// Device/Application/Bausteine/SMB2_Client/NTLM/Functions/ProcessChallengeMessage
FUNCTION_BLOCK ProcessChallengeMessage
VAR_INPUT
	xExecute:BOOL; // Start
	session:POINTER TO SessionData; // NTLM Parameter
	challMess:POINTER TO CHALLENGE_MESSAGE; // Challenge Message
END_VAR
VAR_OUTPUT
	xDone:BOOL;
END_VAR
VAR
	timestamp:ARRAY[0..7] OF BYTE:= [ 16#C2,16#E8,16#2C,16#F5,16#9C,16#6D,16#D3,16#01];
	step:INT;
	clientChall:ARRAY[0..7] OF BYTE:= [16#bf, 16#c5, 16#f2, 16#3e, 16#c8, 16#82, 16#ba, 16#f1];//[16#9E, 16#B9, 16#86, 16#EC, 16#C3, 16#FE, 16#0F, 16#72]; //[16#87, 16#05, 16#42, 16#8E, 16#2A, 16#A3, 16#5D, 16#26];
	servertest:ARRAY[0..7] OF BYTE:= [16#0E, 16#CB, 16#9E, 16#63, 16#6E, 16#3E, 16#08, 16#50];
	NTOWFv2:NTOWFv2;
	LMOWFv2:LMOWFv2;
	SIGNKEY:SIGNKEY;
	SEALKEY:SEALKEY;
	mechListMic:mechListMic;
	ComputeResponse:ComputeResponse;
END_VAR

// Compute the whole Challenge Message and copy all results to session

xDone:=FALSE;
if step=0 and xExecute then
	step:=1;
END_IF

CASE step OF
1:	session^.serverChallenge := challMess^.ServerChallenge;
	session^.clientChallenge := clientChall;
	session^.NegotiateFlags := 16#E2880215;//challMess^.NegotiateFlags;
	step:=2;
	
	// Response Keys
2:	NTOWFv2(Passwd:=session^.password,User:=session^.user,UserDom:=session^.userDomain,out=>session^.responseKeyNT);
	NTOWFv2.xExecute:= TRUE;
	IF NTOWFv2.xDone THEN step:=step+1; END_IF
3:	LMOWFv2(Passwd:=session^.password,User:=session^.user,UserDom:=session^.userDomain,out=>session^.responseKeyLM);
	LMOWFv2.xExecute:= TRUE;
	IF LMOWFv2.xDone THEN step:=step+1; END_IF

	// Timestamp from Challenge Message
4: 	timestamp:= challMess^.AVPairList.TimeStamp;
	//challMess^.AVPairList.TimeStamp:=timestamp;
	step:=step+1;
	
5:	ComputeResponse(session:=session,challMess:=challMess,Timee:=timeStamp); // Compute NTProofStr, lmResponse, ntResponse, session base key
	ComputeResponse.xExecute:=TRUE;
	IF ComputeResponse.xDone THEN step:=step+1; END_IF

	// KeyExchange Key
6:	session^.keyExchangeKey:= session^.sessionBaseKey;
	step:=step+1;

7: 	// Encrypted Session Key
	EncryptedSessionKey(session:=session);
	step:=step+1;
	
	// Sign & Seal Keys
8:	SIGNKEY(ExportedSessionKey:=session^.exportedSessionKey,NegFlg:=session^.NegotiateFlags,Mode:=1,SignKey=>session^.ClientSigningKey);
	SIGNKEY.xExecute:=TRUE;
	IF SIGNKEY.xDone THEN SIGNKEY.xExecute:=FALSE; step:=step+1; END_IF
	
9:	SIGNKEY(ExportedSessionKey:=session^.exportedSessionKey,NegFlg:=session^.NegotiateFlags,Mode:=2,SignKey=>session^.ServerSigningKey);
	SIGNKEY.xExecute:=TRUE;
	IF SIGNKEY.xDone THEN SIGNKEY.xExecute:=FALSE; step:=step+1; END_IF
	
10:	SEALKEY(ExportedSessionKey:=session^.exportedSessionKey,NegFlg:=session^.NegotiateFlags,Mode:=1,SealKey=>session^.ClientSealingKey);
	SEALKEY.xExecute:=TRUE;
	IF SEALKEY.xDone THEN SEALKEY.xExecute:=FALSE; step:=step+1; END_IF
	
11:	SEALKEY(ExportedSessionKey:=session^.exportedSessionKey,NegFlg:=session^.NegotiateFlags,Mode:=2,SealKey=>session^.ServerSealingKey);
	SEALKEY.xExecute:=TRUE;
	IF SEALKEY.xDone THEN SEALKEY.xExecute:=FALSE; step:=step+1; END_IF

12:	mechListMic(session:=session,out=>session^.mechListMIC);
	mechListMic.xExecute:=TRUE;
	IF mechListMic.xDone THEN SEALKEY.xExecute:=FALSE; step:=step+1; END_IF
	
	// RC4 Init
13:	session^.clientHandle(key:=ADR(session^.ClientSealingKey),lenKey:=16,Mode:=0);
	session^.ServerHandle(key:=ADR(session^.ServerSealingKey),lenKey:=16,Mode:=0);
	xDone:=TRUE;
	step:=0;
	
END_CASE

END_FUNCTION_BLOCK

// Device/Application/Bausteine/SMB2_Client/NTLM/Functions/NTOWFv2
FUNCTION_BLOCK NTOWFv2
VAR_INPUT
	xExecute:BOOL;
	Passwd:WSTRING;
	User:WSTRING;
	UserDom:WSTRING;
END_VAR
VAR_OUTPUT
	xDone:BOOL;
	out:ARRAY[0..15] OF BYTE;
END_VAR
VAR
	Step:INT:=0;
	temp:ARRAY[0..15] OF BYTE:= [16#DD, 16#D0,16#B7,16#46,16#5E,16#B8,16#39,16#32,16#66,16#98,16#3F,16#B8,16#4D,16#7B,16#AD,16#9D];;
	concat:WSTRING;
	MD4:MD4;
	HMACMD5:HMAC_MD5;
END_VAR

(*
[MS-NLMP]
NTOWFv2(Passwd, User, UserDom) as HMAC_MD5( MD4(UNICODE(Passwd)), UNICODE(ConcatenationOf( Uppercase(User), UserDom ) ) )
*)

xDone := FALSE;
IF Step = 0 AND xExecute = 1 THEN
	Step:=1;
END_IF

CASE Step OF
0: 	xDone := FALSE;

1:	MD4(PT:=ADR(Passwd),Length:=(WLEN(Passwd)*2),digest=>temp); //MD4(UNICODE(Passwd))
	concat:= WCONCAT(WSTRING_UPPER(User),UserDom); // UNICODE(ConcatenationOf( Uppercase(User), UserDom )
	Step := 2;
	
2:	HMACMD5(key:=ADR(temp),lenKey:=16,message:=ADR(concat),lenMess:=WLEN(concat)*2,out=>out); // Hash HMAC_MD5( MD4(UNICODE(Passwd)), UNICODE(ConcatenationOf( Uppercase(User), UserDom ) ) )
	HMACMD5.xExecute:= TRUE;
	
	IF HMACMD5.xDone THEN
		HMACMD5.xExecute:= TRUE;	
		xDone := TRUE;
		Step:=0;
	END_IF
END_CASE

END_FUNCTION_BLOCK

// Device/Application/Bausteine/SMB2_Client/NTLM/Functions/Hash/Encryption/MD4
FUNCTION_BLOCK MD4
VAR_INPUT
	PT: POINTER TO ARRAY[0..127]OF BYTE;
	Length:INT;
END_VAR
VAR_OUTPUT
	digest:ARRAY[0..15] OF byte;
END_VAR
VAR
	A:UDINT:= 16#67452301;
	AA:UDINT:=0;
	B:UDINT:= 16#EFCDAB89; 
	BB:UDINT:=0;
	C:UDINT:= 16#98BADCFE; 
	CC:UDINT:=0;
	D:UDINT:= 16#10325476;
	DD:UDINT:=0;
	i:INT;
	j:INT;
	M:ARRAY[0..127] OF BYTE;
	MM:ARRAY[0..31] OF UDINT;
	X:ARRAY[0..15] OF UDINT;
	Len:INT;
	pVar:POINTER TO ARRAY[0..127] OF BYTE;
	pVar2:POINTER TO BYTE;
END_VAR

	A:=16#67452301;
	B:= 16#EFCDAB89; 
	C:= 16#98BADCFE; 
	D:= 16#10325476;
	
FOR i:=0 TO Length-1 DO
	M[i]:= PT^[i];
END_FOR
	// Apped 1 Bit to the Message
	M[Length] := 16#80;
	
	pVar:=ADR(M[0]);
	pVar2:=ADR(MM[0]);
	FOR i:=0 TO ((len+1)*64)-1 DO
		pVar2^:=pVar^[i];
		pVar2:=pVar2+1;
	END_FOR
	
	
IF Length < 64 THEN
	MM[14]:= INT_TO_UDINT(Length*8);
	len:=0;
ELSIF Length >= 64 AND Length < 128 THEN
	MM[30]:= INT_TO_UDINT(Length*8);
	len:=1;
END_IF	

	
FOR i:=0 TO len DO
	// Copy block i into X
	FOR j:=0 TO 15 DO
		X[j]:= MM[16*i+j];
	END_FOR
	 
	AA:=A;
	BB:=B;
	CC:=C;
	DD:=D;
	
	A:= ROUND1(A,B,C,D,X[0],3);
	D:=	ROUND1(D,A,B,C,X[1],7);
	C:=	ROUND1(C,D,A,B,X[2],11);
	B:=	ROUND1(B,C,D,A,X[3],19);
	A:=	ROUND1(A,B,C,D,X[4],3);
	D:=	ROUND1(D,A,B,C,X[5],7);
	C:=	ROUND1(C,D,A,B,X[6],11);
	B:=	ROUND1(B,C,D,A,X[7],19);
	A:=	ROUND1(A,B,C,D,X[8],3);
	D:=	ROUND1(D,A,B,C,X[9],7);
	C:=	ROUND1(C,D,A,B,X[10],11);
	B:=	ROUND1(B,C,D,A,X[11],19);
	A:=	ROUND1(A,B,C,D,X[12],3);
	D:=	ROUND1(D,A,B,C,X[13],7);
	C:=	ROUND1(C,D,A,B,X[14],11);
	B:=	ROUND1(B,C,D,A,X[15],19);
	
	A:=	ROUND2(A,B,C,D,X[0],3);
	D:=	ROUND2(D,A,B,C,X[4],5);
	C:=	ROUND2(C,D,A,B,X[8],9);
	B:=	ROUND2(B,C,D,A,X[12],13);
	A:=	ROUND2(A,B,C,D,X[1],3);
	D:=	ROUND2(D,A,B,C,X[5],5);
	C:=	ROUND2(C,D,A,B,X[9],9);
	B:=	ROUND2(B,C,D,A,X[13],13);
	A:=	ROUND2(A,B,C,D,X[2],3);
	D:=	ROUND2(D,A,B,C,X[6],5);
	C:=	ROUND2(C,D,A,B,X[10],9);
	B:=	ROUND2(B,C,D,A,X[14],13);
	A:=	ROUND2(A,B,C,D,X[3],3);
	D:=	ROUND2(D,A,B,C,X[7],5);
	C:=	ROUND2(C,D,A,B,X[11],9);
	B:=	ROUND2(B,C,D,A,X[15],13);
 
	A:=	ROUND3(A,B,C,D,X[0],3);
	D:=	ROUND3(D,A,B,C,X[8],9);
	C:=	ROUND3(C,D,A,B,X[4],11);
	B:=	ROUND3(B,C,D,A,X[12],15);
	A:=	ROUND3(A,B,C,D,X[2],3);
	D:=	ROUND3(D,A,B,C,X[10],9);
	C:=	ROUND3(C,D,A,B,X[6],11);
	B:=	ROUND3(B,C,D,A,X[14],15);
	A:=	ROUND3(A,B,C,D,X[1],3);
	D:=	ROUND3(D,A,B,C,X[9],9);
	C:=	ROUND3(C,D,A,B,X[5],11);
	B:=	ROUND3(B,C,D,A,X[13],15);
	A:=	ROUND3(A,B,C,D,X[3],3);
	D:=	ROUND3(D,A,B,C,X[11],9);
	C:=	ROUND3(C,D,A,B,X[7],11);
	B:=	ROUND3(B,C,D,A,X[15],15);
	
	A:=A+AA;
	B:=B+BB;
	C:=C+CC;
	D:=D+DD;
END_FOR

	digest[0]:=UDINT_TO_BYTE(A); digest[1]:=UDINT_TO_BYTE(SHR(A,8)); digest[2]:=UDINT_TO_BYTE(SHR(A,16)); digest[3]:=UDINT_TO_BYTE(SHR(A,24)); 
	digest[4]:=UDINT_TO_BYTE(B); digest[5]:=UDINT_TO_BYTE(SHR(B,8)); digest[6]:=UDINT_TO_BYTE(SHR(B,16)); digest[7]:=UDINT_TO_BYTE(SHR(B,24)); 
	digest[8]:=UDINT_TO_BYTE(C); digest[9]:=UDINT_TO_BYTE(SHR(C,8)); digest[10]:=UDINT_TO_BYTE(SHR(C,16)); digest[11]:=UDINT_TO_BYTE(SHR(C,24)); 
	digest[12]:=UDINT_TO_BYTE(D); digest[13]:=UDINT_TO_BYTE(SHR(D,8)); digest[14]:=UDINT_TO_BYTE(SHR(D,16)); digest[15]:=UDINT_TO_BYTE(SHR(D,24)); 

FOR i:=0 TO 127 DO
	M[i] := 0;
END_FOR

METHOD ROUND1 : UDINT
VAR_INPUT
	a:UDINT;
	b:UDINT;
	c:UDINT;
	d:UDINT;
	x:UDINT;
	ss:UDINT;
END_VAR
VAR
	temp:UDINT;
	temp1:UDINT;
	temp2:udint;
END_VAR
//#define F(X,Y,Z) (((X)&(Y))|((~(X))&(Z)))
//#define G(X,Y,Z) (((X)&(Y))|((X)&(Z))|((Y)&(Z)))
//#define H(X,Y,Z) ((X)^(Y)^(Z))
 
//#define LEFTROTATE(A,N) ((A)<<(N))|((A)>>(32-(N)))
 
//#define MD4ROUND1(a,b,c,d,x,s) a += F(b,c,d) + x; a = LEFTROTATE(a, s);
//#define MD4ROUND2(a,b,c,d,x,s) a += G(b,c,d) + x + (uint32_t)0x5A827999; a = LEFTROTATE(a, s);
//#define MD4ROUND3(a,b,c,d,x,s) a += H(b,c,d) + x + (uint32_t)0x6ED9EBA1; a = LEFTROTATE(a, s);

temp:= a  ;
temp1:=(((b AND c) OR ((NOT b) AND d))) ;
temp2:= x;

temp1:= temp+temp1;
temp:= temp1 + temp2;
ROUND1:= ROL(temp, ss);
END_METHOD

METHOD ROUND2 : UDINT
VAR_INPUT
	a:UDINT;
	b:UDINT;
	c:UDINT;
	d:UDINT;
	x:UDINT;
	ss:UDINT;
END_VAR
VAR
	temp:UDINT;
END_VAR
//#define F(X,Y,Z) (((X)&(Y))|((~(X))&(Z)))
//#define G(X,Y,Z) (((X)&(Y))|((X)&(Z))|((Y)&(Z)))
//#define H(X,Y,Z) ((X)^(Y)^(Z))
 
//#define LEFTROTATE(A,N) ((A)<<(N))|((A)>>(32-(N)))
 
//#define MD4ROUND1(a,b,c,d,x,s) a += F(b,c,d) + x; a = LEFTROTATE(a, s);
//#define MD4ROUND2(a,b,c,d,x,s) a += G(b,c,d) + x + (uint32_t)0x5A827999; a = LEFTROTATE(a, s);
//#define MD4ROUND3(a,b,c,d,x,s) a += H(b,c,d) + x + (uint32_t)0x6ED9EBA1; a = LEFTROTATE(a, s);

temp:= a + (((b)AND(c))OR((b)AND(d))OR((c)AND(d))) + x + 16#5A827999;

ROUND2:= ROL(temp, ss);
END_METHOD

METHOD ROUND3 : UDINT
VAR_INPUT
	a:UDINT;
	b:UDINT;
	c:UDINT;
	d:UDINT;
	x:UDINT;
	ss:UDINT;
END_VAR
VAR
	temp:UDINT;
END_VAR
//#define F(X,Y,Z) (((X)&(Y))|((~(X))&(Z)))
//#define G(X,Y,Z) (((X)&(Y))|((X)&(Z))|((Y)&(Z)))
//#define H(X,Y,Z) ((X)^(Y)^(Z))
 
//#define LEFTROTATE(A,N) ((A)<<(N))|((A)>>(32-(N)))
 
//#define MD4ROUND1(a,b,c,d,x,s) a += F(b,c,d) + x; a = LEFTROTATE(a, s);
//#define MD4ROUND2(a,b,c,d,x,s) a += G(b,c,d) + x + (uint32_t)0x5A827999; a = LEFTROTATE(a, s);
//#define MD4ROUND3(a,b,c,d,x,s) a += H(b,c,d) + x + (uint32_t)0x6ED9EBA1; a = LEFTROTATE(a, s);

temp:= a + ((b)XOR(c)XOR(d)) + x + 16#6ED9EBA1;

ROUND3:= ROL(temp, ss);
END_METHOD

END_FUNCTION_BLOCK

// Device/Application/Bausteine/SMB2_Client/Misc/WSTRING_UPPER
FUNCTION WSTRING_UPPER : WSTRING(80)
VAR_INPUT
	In:WSTRING(80);
END_VAR
VAR
	i:int;
	len:INT;
	pIn:POINTER TO ARRAY[0..79] OF WORD;
	pOut:POINTER TO ARRAY[0..79] OF WORD;
END_VAR

len:=wlen(In);

pIn:= ADR(In);
pOut:= ADR(WSTRING_UPPER);

FOR i:=0 TO len DO
	IF pIn^[i] >= 16#0061 AND pIn^[i] <= 16#007A THEN
		pOut^[i] := pIn^[i] - 16#0020;
	ELSE
		pOut^[i]:=pIn^[i]; 
	END_IF
END_FOR

END_FUNCTION

// Device/Application/Bausteine/SMB2_Client/NTLM/Functions/LMOWFv2
FUNCTION_BLOCK LMOWFv2
VAR_INPUT
	xExecute:BOOL;
	Passwd:WSTRING;
	User:WSTRING;
	UserDom:WSTRING;
END_VAR
VAR_OUTPUT
	xDone:BOOL;
	out:ARRAY[0..15] OF BYTE;
END_VAR
VAR
	NTOWFv2:NTOWFv2;
END_VAR

(*
[MS-NLMP]
LMOWFv2(Passwd, User, UserDom) as NTOWFv2(Passwd, User, UserDom)
*)

NTOWFv2(xExecute:= xExecute,Passwd:=Passwd,User:=User,UserDom:=UserDom,xDone=>xDone,out=>out);

END_FUNCTION_BLOCK

// Device/Application/Bausteine/SMB2_Client/NTLM/Functions/ComputeResponse
FUNCTION_BLOCK ComputeResponse
VAR_INPUT
	xExecute:BOOL; // Start
	session:POINTER TO sessionData; // NTLM Parameter
	challMess:POINTER TO CHALLENGE_MESSAGE; // Challenge Message
	Timee:ARRAY[0..7] OF BYTE; // Timestamp from Challenge Message
END_VAR
VAR_OUTPUT
	xDone:BOOL;
END_VAR
VAR
	Step:INT:=0;
	i:INT;
	temp:ARRAY[0..511] OF BYTE;
	tempLen:INT;
	pVar:POINTER TO ARRAY[0..32767] OF BYTE;
	ntProofStr:ARRAY[0..15] OF BYTE;
	temp2:ARRAY[0..511] OF BYTE;
	tempLen2:INT;
	hmacTemp:ARRAY[0..15] OF BYTE;
	HMACMD5:HMAC_MD5;

END_VAR

(*
	[MS-NLMP]
	Set temp to ConcatenationOf(Responserversion, HiResponserversion, Z(6), Time, ClientChallenge, Z(4), ServerName, Z(4)) 
	Set NTProofStr to HMAC_MD5(ResponseKeyNT, ConcatenationOf(CHALLENGE_MESSAGE.ServerChallenge,temp)) 
	Set NtChallengeResponse to ConcatenationOf(NTProofStr, temp) 
	Set LmChallengeResponse to ConcatenationOf(HMAC_MD5(ResponseKeyLM, ConcatenationOf(CHALLENGE_MESSAGE.ServerChallenge, ClientChallenge)), ClientChallenge )
*)

xDone:=FALSE;
IF Step = 0 AND xExecute = TRUE THEN
	Step:=1;
END_IF

CASE step OF
0:	
1:	//ConcatenationOf(Responserversion, HiResponserversion, Z(6), Time, ClientChallenge, Z(4), AVPairList, Z(4)) // Servername in NLMP Kap 3.3.1 means AVPairList
	i:=0;
	pVar:=ADR(temp);
	
	tempLen2 :=SetAVPairList(AVPairList:=challMess^.AVPairList,pOut:=ADR(temp2));
	
	FOR i:=0 TO 1 DO
		pVar^[i]:= 16#01;
	END_FOR
	FOR i:=i TO 1+6 DO
		pVar^[i]:= 16#00;
	END_FOR
	FOR i:=i TO 1+6+8 DO
		pVar^[i] := timee[i-(1+1+6)];
	END_FOR
	FOR i:=i TO 1+6+8+8 DO
		pVar^[i] :=	session^.clientChallenge[i-(1+1+6+8)];
	END_FOR
	FOR i:=i TO 1+6+8+8+4 DO
		pVar^[i]:= 16#00;
	END_FOR
	FOR i:=i TO 1+6+8+8+4+tempLen2 DO
		pVar^[i]:= temp2[i-(1+1+6+8+8+4)];
	END_FOR
	FOR i:=i TO 1+6+8+8+4+tempLen2+4 DO
		pVar^[i]:= 16#00;
	END_FOR
	tempLen:=i;
	step:=step+1;
	
	// ConcatenationOf(serverchallenge, temp)
2:	FOR i:=0 TO 7 DO
		temp2[i] := session^.serverChallenge[i];
	END_FOR
	FOR i:=i TO 7+tempLen DO
		temp2[i] := temp[i-(1+7)];
	END_FOR
	tempLen2:=i;
	step:=step+1;
	
	// NTProofStr = HMAC_MD5(responseKeyNt, temp2)
3:	HMACMD5(key:=ADR(session^.responseKeyNT),lenKey:=16 ,message:=ADR(temp2[0]), lenMess:=tempLen2+4,out=>ntProofStr); //<-- +4
	HMACMD5.xExecute:= TRUE;
	
	IF HMACMD5.xDone THEN
		step:= 4;
		HMACMD5.xExecute:= FALSE;
	END_IF

	// ntChallengeResponse = concat(ntProofStr, temp)
4:	FOR i:=0 TO 15 DO
		session^.ntChallengeResponse[i] := ntProofStr[i];
	END_FOR
	FOR i:=i TO 15+tempLen DO
		session^.ntChallengeResponse[i] := temp[i-(1+15)];
	END_FOR
	session^.ntChallengeResponseLen := INT_TO_WORD(i)+4; //<-- +4
	step:=step+1;
	
	// n.lmChallengeResponse = concat(hmacMd5(n.responseKeyLM, concat(n.serverChallenge, n.clientChallenge)), n.clientChallenge)
5:	FOR i:=0 TO 7 DO
		temp2[i] := session^.serverChallenge[i];
	END_FOR
	FOR i:=i TO 7+8 DO
		temp2[i] := session^.clientChallenge[i-8];
	END_FOR
	step:=step+1;
	
6: 	HMACMD5(key:=ADR(session^.responseKeyLM),lenKey:=16 ,message:=ADR(temp2[0]), lenMess:=32,out=>hmacTemp);
	HMACMD5.xExecute:= TRUE;
	
	IF HMACMD5.xDone THEN
		step:= 7;
		HMACMD5.xExecute:= FALSE;
	END_IF
	
7:	// Concat lmChallengeResponse
	FOR i:=0 TO 15 DO
		session^.lmChallengeResponse[i] := hmacTemp[i];
	END_FOR
	FOR i:=i TO 15+8 DO
		session^.lmChallengeResponse[i] := session^.clientChallenge[i-15];
	END_FOR
	session^.lmChallengeResponseLen := INT_TO_WORD(i);
	step:=step+1;
	FOR i:=0 TO UINT_TO_INT(session^.lmChallengeResponseLen) -1 DO // Make lmChallengeResponse zero, not used
		session^.lmChallengeResponse[i]:= 0;
	END_FOR
	
	
	// sessionBaseKey = hmacMd5(responseKeyNT, ntProofStr)
8: 	HMACMD5(key:=ADR(session^.responseKeyNT),lenKey:=16 ,message:=ADR(ntProofStr[0]), lenMess:=16,out=>session^.sessionBaseKey);
	HMACMD5.xExecute:= TRUE;
	
	IF HMACMD5.xDone THEN
		step:= 0;
		HMACMD5.xExecute:= FALSE;
		xDone:=TRUE;
	END_IF
END_CASE

END_FUNCTION_BLOCK

// Device/Application/Bausteine/SMB2_Client/NTLM/Functions/SetAVPairList
FUNCTION SetAVPairList : int
VAR_INPUT
	AVPairList:AVPairList; // Extracted Attribute from Challenge Message
	pOut:POINTER TO ARRAY[0..32767] OF BYTE; // Pointer to Buffer or Payload Buffer
END_VAR
VAR
	step:INT:=1;
	pVar:POINTER TO ARRAY[0..511] OF BYTE;
	pVarLen:POINTER TO ARRAY[0..511] OF BYTE;
	i:INT:=0;
	j:INT:=0;
	tempLen:INT;
	identifier:BYTE;;
	flags:DWORD:=16#00000002;
	channelBindings:ARRAY[0..15] OF BYTE:=[0];
	restrictions:ARRAY[0..47] OF BYTE:=	[16#30, 16#00, 16#00, 16#00, 16#00, 16#00, 16#00, 16#00, 16#01, 16#00, 16#00, 16#00, 16#00, 16#20, 16#00, 16#00,
										16#1C, 16#3A, 16#00, 16#6B, 16#51, 16#EA, 16#FC, 16#D1, 16#83, 16#AE, 16#BE, 16#D7, 16#48, 16#1C, 16#34, 16#4D,
										16#1C, 16#13, 16#C4, 16#E4, 16#4C, 16#39, 16#E8, 16#B8, 16#05, 16#4C, 16#63, 16#41, 16#66, 16#FF, 16#57, 16#0D];
	target:WSTRING(80);
	cifs:WSTRING:="cifs/";
	endOfList:BOOL;
END_VAR

// Building a new AVPairList / Target Info for Auth Message

endOfList:=0;
WHILE endOfList = 0 DO
	CASE step OF
		
		1:	// NB Domain Name
			tempLen :=wlen(AVPairList.NBDomainName)*2;
			pVar := ADR(AVPairList.NBDomainName);
			identifier:= 16#02;
			step:=step+1;
		2:	// NB Computer Name
			tempLen :=wlen(AVPairList.NBComputerName)*2;
			pVar := ADR(AVPairList.NBComputerName);
			identifier:= 16#01;
			step:=step+1;
		3:	// DNS Domain Name
			tempLen :=wlen(AVPairList.DNSDomainName)*2;
			pVar := ADR(AVPairList.DNSDomainName);
			identifier:= 16#04;
			step:=step+1;
		4:	// DNS Computer Name
			tempLen :=wlen(AVPairList.DNSComputerName)*2;
			pVar := ADR(AVPairList.DNSComputerName);
			identifier:= 16#03;
			step:=step+1;
		5:	// Timestamp
			tempLen :=8;
			pVar := ADR(AVPairList.TimeStamp);
			identifier:= 16#07;
			step:=step+1;
		6:	// Flags
			tempLen :=4;
			pVar := ADR(flags);
			identifier:= 16#06;
			step:=step+1;
		7:	// Restrictions
			tempLen := 48;
			pVar := ADR(restrictions);
			identifier:= 16#08;
			step:=step+1;
		8:	// Channel Bindings
			tempLen :=16;
			pVar := ADR(channelBindings);
			identifier:= 16#0A;
			step:=step+1;
		9:	// Target Name
			target:=wconcat(cifs,AVPairList.NBComputerName);
			tempLen :=wlen(target)*2;
			pVar := ADR(target);
			identifier:= 16#09;
			step:=1;
			// End of List
			endOfList:=TRUE;
	END_CASE
	// Identifier 
	pOut^[i]:= identifier; pOut^[i+1]:= 16#00; 
	i:=i+2;
	// length
	pVarLen := ADR(tempLen);
	FOR j:=0 TO 1 DO
		pOut^[i] := pVarLen ^[j];
		i:=i+1;
	END_FOR
	// data
	FOR j:=0 TO tempLen-1 DO
		pOut^[i] := pVar^[j];
		i:=i+1;
	END_FOR
	
	IF endOfList THEN
		FOR j:=0 TO 3 DO
		pOut^[i] := 16#00;
		i:=i+1;
		END_FOR
		SetAVPairList:=i;
	END_IF
END_WHILE

END_FUNCTION

// Device/Application/Bausteine/SMB2_Client/NTLM/Functions/EncryptedSessionKey
FUNCTION EncryptedSessionKey : int
VAR_INPUT
	session:POINTER TO sessionData;
END_VAR
VAR
	i:INT;
	temp:ARRAY[0..15] OF BYTE:=[16#C7, 16#9A, 16#31, 16#B6, 16#8D, 16#B6, 16#4E, 16#3F, 16#84, 16#66, 16#BE, 16#A3, 16#B2, 16#22, 16#3B, 16#C1];
	RC4K:RC4;
	temp2:dword;
END_VAR

(*	[MS-NLMP]
	If (NTLMSSP_NEGOTIATE_KEY_EXCH flag is set in NegFlg AND (NTLMSSP_NEGOTIATE_SIGN OR NTLMSSP_NEGOTIATE_SEAL are set in NegFlg) ) 
		Set ExportedSessionKey to RC4K(KeyExchangeKey, AUTHENTICATE_MESSAGE.EncryptedRandomSessionKey) 
	Else 
		Set ExportedSessionKey to KeyExchangeKey 
	EndIf 
*)

	temp2:= session^.NegotiateFlags AND 16#40000000;
IF (session^.NegotiateFlags AND 16#40000000) = 16#40000000 THEN
	session^.exportedSessionKey:= temp;
	RC4K(key:=ADR(session^.keyExchangeKey),lenKey:=16,data:=ADR(session^.exportedSessionKey),lenData:=16,ciper:=ADR(session^.encryptedRandomSessionKey),Mode:=2);
ELSE
	session^.exportedSessionKey := session^.keyExchangeKey;
	FOR i:=0 TO 15 DO
		session^.encryptedRandomSessionKey[i] := 16#00;
	END_FOR
END_IF

END_FUNCTION

// Device/Application/Bausteine/SMB2_Client/NTLM/Functions/SIGNKEY
FUNCTION_BLOCK SIGNKEY
VAR_INPUT
	xExecute:BOOL; // Start
	ExportedSessionKey:ARRAY[0..15] OF BYTE; // Exported Session Key
	NegFlg:DWORD; // Negotiate Flags
	Mode:BYTE; // 1= Client Signing Key, 2= Server Signing Key
END_VAR
VAR_OUTPUT
	xDone:BOOL;
	SignKey:ARRAY[0..15] OF BYTE;
END_VAR
VAR
	Step:INT;
	pVar:POINTER TO ARRAY[0..255] OF BYTE;
	i:INT;
	temp:ARRAY[0..74] OF BYTE;
	hash: MEM.MD5;
END_VAR
VAR CONSTANT
	Client:STRING:='session key to client-to-server signing key magic constant';
	Server:STRING:='session key to server-to-client signing key magic constant';
END_VAR

// This Function generates the Signing key from ExportedSessionKey and static String

//MS-NLMP 3.4.5.2

IF Step = 0 AND xExecute = TRUE THEN
	Step:=1;
ELSE
	xDone:= FALSE;
END_IF

IF (NegFlg AND UDINT_TO_DWORD(16#00080000)) = 16#00080000 THEN // EXTENDED_SESSIONSECURITY flag
	IF Mode = 1 THEN
		CASE Step OF
		0:	xDone:= FALSE;
		1:	FOR i:=0 TO 15 DO
				temp[i]:= ExportedSessionKey[i];
			END_FOR
			pVar:= ADR(Client);
			FOR i:=16 TO 16+standard.LEN(Client) DO
				temp[i]:= pVar^[i-16];
			END_FOR
				temp[i]:=0;
			Step:=2;
		2:	hash(pMemoryBlock:=ADR(Temp[0]),udiNumberOfBytes:=INT_TO_UDINT(16+standard.LEN(Client)+1),abyDigest=>SignKey);
			hash.xExecute:= TRUE;
	
			IF hash.xDone THEN
				step:= 0;
				hash.xExecute:= FALSE;
				xDone:= TRUE;
			END_IF
		END_CASE
	END_IF
	IF Mode = 2 THEN
		CASE Step OF
		0:	xDone:= FALSE;
		1:	FOR i:=0 TO 15 DO
				temp[i]:= ExportedSessionKey[i];
			END_FOR
			pVar:= ADR(Server);
			FOR i:=16 TO 16+standard.LEN(Server) DO
				temp[i]:= pVar^[i-16];
			END_FOR
			temp[i]:=0;
			Step:=2;
		2:	hash(pMemoryBlock:=ADR(Temp[0]),udiNumberOfBytes:=INT_TO_UDINT(standard.LEN(Client)+16+1),abyDigest=>SignKey);
			hash.xExecute:= TRUE;
	
			IF hash.xDone THEN
				step:= 0;
				hash.xExecute:= FALSE;
				xDone:= TRUE;
			END_IF
		END_CASE
	END_IF
ELSE
	FOR i:=0 TO 15 DO
		SignKey[i]:=0;	
	END_FOR
	xDone:= TRUE;
END_IF

END_FUNCTION_BLOCK

// Device/Application/Bausteine/SMB2_Client/NTLM/Functions/SEALKEY
FUNCTION_BLOCK SEALKEY
VAR_INPUT
	xExecute:BOOL; // Start
	ExportedSessionKey:ARRAY[0..15] OF BYTE; // Exported Session Key
	NegFlg:DWORD; // Negotiate Flags
	Mode:BYTE; // 1= Client Sealing Key, 2= Server Sealing Key
END_VAR
VAR_OUTPUT
	xDone:BOOL;
	SealKey:ARRAY[0..15] OF BYTE;
END_VAR
VAR
	SealKeyLen:INT;
	Step:INT;
	pVar:POINTER TO ARRAY[0..255] OF BYTE;
	i:INT;
	temp:ARRAY[0..74] OF BYTE;
	hash: MEM.MD5;
END_VAR
VAR CONSTANT
	Client:STRING:='session key to client-to-server sealing key magic constant';
	Server:STRING:='session key to server-to-client sealing key magic constant';
END_VAR

// This Function generates the Sealkey from ExportedSessionKey and static String

//MS-NLMP 3.4.5.3

xDone:= FALSE;
IF Step = 0 AND xExecute = TRUE THEN
	Step:=1;
END_IF


IF (NegFlg AND UDINT_TO_DWORD(16#00080000)) = 16#00080000 THEN // EXTENDED_SESSIONSECURITY flag
	IF (NegFlg AND UDINT_TO_DWORD(16#20000000)) = 16#20000000 THEN // NTLMSSP_NEGOTIATE_128
		SealKeyLen:= 16;
	ELSIF (NegFlg AND UDINT_TO_DWORD(16#80000000)) = 16#80000000 THEN // NTLMSSP_NEGOTIATE_56
		SealKeyLen:= 7;
	ELSE 
		SealKeyLen:= 5;
	END_IF

	IF Mode = 1 THEN
		CASE Step OF
		0:	xDone:= FALSE;
		1:	FOR i:=0 TO SealKeyLen DO
				temp[i]:= ExportedSessionKey[i];
			END_FOR
			pVar:= ADR(Client);
			FOR i:=SealKeyLen TO SealKeyLen+standard.LEN(Client) DO
				temp[i]:= pVar^[i-16];
			END_FOR
			temp[i]:=0;
			Step:=2;
		2:	hash(pMemoryBlock:=ADR(Temp[0]),udiNumberOfBytes:=INT_TO_UDINT(SealKeyLen+standard.LEN(Client)+1),abyDigest=>SealKey);
			hash.xExecute:= TRUE;
	
			IF hash.xDone THEN
				step:= 0;
				hash.xExecute:= FALSE;
				xDone:= TRUE;
			END_IF
		END_CASE
	ELSE
		CASE Step OF
		0:	xDone:= FALSE;
		1:	FOR i:=0 TO SealKeyLen DO
				temp[i]:= ExportedSessionKey[i];
			END_FOR
			pVar:= ADR(Server);
			FOR i:=SealKeyLen TO SealKeyLen+standard.LEN(Server) DO
				temp[i]:= pVar^[i-16];
			END_FOR
			temp[i]:=0;
			Step:=2;
		2:	hash(pMemoryBlock:=ADR(Temp[0]),udiNumberOfBytes:=INT_TO_UDINT(SealKeyLen+standard.LEN(Server)+1),abyDigest=>SealKey);
			hash.xExecute:= TRUE;
	
			IF hash.xDone THEN
				step:= 0;
				hash.xExecute:= FALSE;
				xDone:= TRUE;
			END_IF
		END_CASE
	END_IF
ELSIF ((NegFlg AND UDINT_TO_DWORD(16#00000200)) = 16#00000200) OR	// LM KEY
		((NegFlg AND UDINT_TO_DWORD(16#00000040)) = 16#00000040) THEN // DATAGRAM

	IF (NegFlg AND UDINT_TO_DWORD(16#80000000)) = 16#80000000 THEN // NTLMSSP_NEGOTIATE_56
		FOR i:=0 TO 5 DO
			temp[i]:= ExportedSessionKey[i];
		END_FOR
		temp[7]:= 16#A0;
	ELSE
		FOR i:=0 TO 4 DO
			temp[i]:= ExportedSessionKey[i];
		END_FOR
		temp[5]:= 16#E5; temp[6]:= 16#38; temp[7]:= 16#B0;
	END_IF
	FOR i:=0 TO 15 DO
		SealKey[i]:=temp[i];	
	END_FOR
	Step:=0;
	xDone:= TRUE;
ELSE
	FOR i:=0 TO 15 DO
		SealKey[i]:=ExportedSessionKey[i];	
	END_FOR
	Step:=0;
	xDone:= TRUE;
END_IF

END_FUNCTION_BLOCK

// Device/Application/Bausteine/SMB2_Client/SMB2/Functions/Requests/TreeConnectReq
FUNCTION TreeConnectReq : int
VAR_INPUT
	Connection:POINTER TO Connection; // Connection Parameter
	pSend:POINTER TO ARRAY[0..32767] OF BYTE; // Pointer to Send Buffer
	pSize:POINTER TO CAA.SIZE; // Send Size
	SharePathName:WSTRING(256); // name of Sharepath
END_VAR
VAR
	TransportHeader:SMB2_Transport_Header;
	SMB2Header: SMB2_Header_Sync;
	SMB2TreeConnect:SMB2_TREE_CONNECT_Request;
	sendS:UINT;
	startIndex:UINT;
END_VAR

// This Function generates the Tree Connect Request

	// Increase Message ID
	Connection^.MessageID[0]:= Connection^.MessageID[0]+1;	
	// Create Header
	SMB2Header.ProtocolID[0]:= 16#FE; SMB2Header.ProtocolID[1]:= 16#53; SMB2Header.ProtocolID[2]:= 16#4D; SMB2Header.ProtocolID[3]:= 16#42; 
	SMB2Header.StructureSize := 64;
	SMB2Header.CreditCharge := 0;
	SMB2Header.Status := 0;
	SMB2Header.Command := Constants.TREE_CONNECT;
	SMB2Header.CreditRepReq := 1;
	SMB2Header.Flags:= 0;
	SMB2Header.Flags := 0;
	SMB2Header.NextCommand := 0;		
	SMB2Header.MessageID[0]:= Connection^.MessageID[0]; SMB2Header.MessageID[1]:= 0;
	SMB2Header.TreeID:= 0;
	SMB2Header.SessionID[0]:= Connection^.Session.SessionID[0]; SMB2Header.SessionID[1]:= Connection^.Session.SessionID[1];
	SMB2Header.Signature[0]:= 0; SMB2Header.Signature[1]:= 0; SMB2Header.Signature[2]:= 0; SMB2Header.Signature[3]:= 0;
	
	// Create Tree Connect Request
	SMB2TreeConnect.StructureSize:= 9;
	SMB2TreeConnect.Flags:=0;
	SMB2TreeConnect.PathOffset:= 64 + 8;
	SMB2TreeConnect.PathName := SharePathName;
	SMB2TreeConnect.PathLength := INT_TO_WORD(wlen(SMB2TreeConnect.PathName)*2);
	
	
	// Copy Data in SendBuffer
	sendS:=SIZEOF(SMB2_Transport_Header);
	(*Parse SMB2 Header*)
	startIndex:=sendS-1;
	sendS:=sendS+SIZEOF(SMB2Header);
	MEM.MemMove(pSource:=ADR(SMB2Header) , pDestination:=ADR(pSend^[startIndex]) ,uiNumberOfBytes:=SIZEOF(SMB2Header));
	
	(*Parse Tree Connect Request*)
	startIndex:=sendS-1;
	sendS:=sendS+WORD_TO_UINT(SMB2TreeConnect.StructureSize-1+SMB2TreeConnect.PathLength);
	MEM.MemMove(pSource:=ADR(SMB2TreeConnect) , pDestination:=ADR(pSend^[startIndex]) ,uiNumberOfBytes:=WORD_TO_UINT(SMB2TreeConnect.StructureSize)-1+SMB2TreeConnect.PathLength);
	
	(*Parse Transport Header*)
	TransportHeader.Zero := 16#00;
	TransportHeader.StreamProtocolLength := SHR(MEM.ReverseBYTEsInDWORD(sendS-SIZEOF(TransportHeader)),8);
		
	startIndex:=0;
	MEM.MemMove(pSource:=ADR(TransportHeader) , pDestination:=ADR(pSend^[startIndex]) ,uiNumberOfBytes:=SIZEOF(SMB2_Transport_Header)-1);
	
	(*Set Sendsize*)	
	pSize^:= sendS-1;

END_FUNCTION

// Device/Application/Bausteine/SMB2_Client/SMB2/Functions/Requests/CloseReq
FUNCTION CloseReq : int
VAR_INPUT
	Connection:POINTER TO Connection; // Connection Parameter
	pSend:POINTER TO ARRAY[0..32767] OF BYTE; // Pointer to Send Buffer
	pSize:POINTER TO CAA.SIZE; // Send Size
END_VAR
VAR
	i:INT;
	TransportHeader:SMB2_Transport_Header;
	SMB2Header: SMB2_Header_Sync;
	SMB2Close: SMB2_Close_Request;
	sendS:UINT;
	startIndex:UINT;
	pVar: POINTER TO ARRAY[0..255] OF BYTE;
END_VAR

// This Function generates the Close Request

	// Increase Message ID
	Connection^.MessageID[0]:= Connection^.MessageID[0]+1;	
	// Create Header
	SMB2Header.ProtocolID[0]:= 16#FE; SMB2Header.ProtocolID[1]:= 16#53; SMB2Header.ProtocolID[2]:= 16#4D; SMB2Header.ProtocolID[3]:= 16#42; 
	SMB2Header.StructureSize := 64;
	SMB2Header.CreditCharge := 0;
	SMB2Header.Status := 0;
	SMB2Header.Command := Constants.CLOSE;
	SMB2Header.CreditRepReq := 1;
	SMB2Header.Flags:= 0;
	SMB2Header.Flags := 0;
	SMB2Header.NextCommand := 0;		
	SMB2Header.MessageID[0]:= Connection^.MessageID[0]; SMB2Header.MessageID[1]:= 0;
	SMB2Header.TreeID:= connection^.Session.TreeConnect.TreeConnectId;
	SMB2Header.SessionID[0]:= Connection^.Session.SessionID[0]; SMB2Header.SessionID[1]:= Connection^.Session.SessionID[1];
	SMB2Header.Signature[0]:= 0; SMB2Header.Signature[1]:= 0; SMB2Header.Signature[2]:= 0; SMB2Header.Signature[3]:= 0;
	
	// Close Request
	SMB2Close.StructureSize := 24;
	SMB2Close.Flags:=0;
	SMB2Close.FileId := Connection[0].Session.Open.FileId;
	
	// Copy Data in SendBuffer
	sendS:=SIZEOF(SMB2_Transport_Header);
	(*Parse SMB2 Header*)
	startIndex:=sendS-1;
	sendS:=sendS+SIZEOF(SMB2Header);
	MEM.MemMove(pSource:=ADR(SMB2Header) , pDestination:=ADR(pSend^[startIndex]) ,uiNumberOfBytes:=SIZEOF(SMB2Header));
	
	(*Parse Close Request*)
	startIndex:=sendS-1;
	sendS:=sendS+WORD_TO_UINT(SMB2Close.StructureSize);
	MEM.MemMove(pSource:=ADR(SMB2Close) , pDestination:=ADR(pSend^[startIndex]) ,uiNumberOfBytes:=WORD_TO_UINT(SMB2Close.StructureSize));
	
	(*Parse Transport Header*)
	TransportHeader.Zero := 16#00;
	TransportHeader.StreamProtocolLength := SHR(MEM.ReverseBYTEsInDWORD(sendS-SIZEOF(TransportHeader)),8);
		
	startIndex:=0;
	MEM.MemMove(pSource:=ADR(TransportHeader) , pDestination:=ADR(pSend^[startIndex]) ,uiNumberOfBytes:=SIZEOF(SMB2_Transport_Header)-1);
	
	(*Set Sendsize*)	
	pSize^:= sendS-1;

END_FUNCTION

// Device/Application/Bausteine/SMB2_Client/SMB2/Functions/Requests/TreeDisconnectReq
FUNCTION TreeDisconnectReq : int
VAR_INPUT
	Connection:POINTER TO Connection; // Connection Parameter
	pSend:POINTER TO ARRAY[0..32767] OF BYTE; // Pointer to Send Buffer
	pSize:POINTER TO CAA.SIZE; // Send Size
END_VAR
VAR
	TransportHeader:SMB2_Transport_Header;
	SMB2Header: SMB2_Header_Sync;
	SMB2Dis: SMB2_TREE_DISCONNECT_Request;
	sendS:UINT;
	startIndex:UINT;
END_VAR

// This Function generates the Tree Disconnect Request

	// Increase Message ID
	Connection^.MessageID[0]:= Connection^.MessageID[0]+1;	
	// Create Header
	SMB2Header.ProtocolID[0]:= 16#FE; SMB2Header.ProtocolID[1]:= 16#53; SMB2Header.ProtocolID[2]:= 16#4D; SMB2Header.ProtocolID[3]:= 16#42; 
	SMB2Header.StructureSize := 64;
	SMB2Header.CreditCharge := 0;
	SMB2Header.Status := 0;
	SMB2Header.Command := Constants.TREE_DISCONNECT;
	SMB2Header.CreditRepReq := 1;
	SMB2Header.Flags:= 0;
	SMB2Header.Flags := 0;
	SMB2Header.NextCommand := 0;		
	SMB2Header.MessageID[0]:= Connection^.MessageID[0]; SMB2Header.MessageID[1]:= 0;
	SMB2Header.TreeID:= connection^.Session.TreeConnect.TreeConnectId;
	SMB2Header.SessionID[0]:= Connection^.Session.SessionID[0]; SMB2Header.SessionID[1]:= Connection^.Session.SessionID[1];
	SMB2Header.Signature[0]:= 0; SMB2Header.Signature[1]:= 0; SMB2Header.Signature[2]:= 0; SMB2Header.Signature[3]:= 0;
	
	// Tree Disconnect Request
	SMB2Dis.StructureSize := 4;
	SMB2Dis.Reserved := 0;
	
	// Copy Data in SendBuffer
	sendS:=SIZEOF(SMB2_Transport_Header);
	(*Parse SMB2 Header*)
	startIndex:=sendS-1;
	sendS:=sendS+SIZEOF(SMB2Header);
	MEM.MemMove(pSource:=ADR(SMB2Header) , pDestination:=ADR(pSend^[startIndex]) ,uiNumberOfBytes:=SIZEOF(SMB2Header));
	
	(*Parse Tree Disconnect Request*)
	startIndex:=sendS-1;
	sendS:=sendS+WORD_TO_UINT(SMB2Dis.StructureSize);
	MEM.MemMove(pSource:=ADR(SMB2Dis) , pDestination:=ADR(pSend^[startIndex]) ,uiNumberOfBytes:=WORD_TO_UINT(SMB2Dis.StructureSize));
	
	(*Parse Transport Header*)
	TransportHeader.Zero := 16#00;
	TransportHeader.StreamProtocolLength := SHR(MEM.ReverseBYTEsInDWORD(sendS-SIZEOF(TransportHeader)),8);
		
	startIndex:=0;
	MEM.MemMove(pSource:=ADR(TransportHeader) , pDestination:=ADR(pSend^[startIndex]) ,uiNumberOfBytes:=SIZEOF(SMB2_Transport_Header)-1);
	
	(*Set Sendsize*)	
	pSize^:= sendS-1;

END_FUNCTION

// Device/Application/Bausteine/SMB2_Client/SMB2/Functions/Requests/LogOffReq
FUNCTION LogOffReq : int
VAR_INPUT
	Connection:POINTER TO Connection; // Connection Parameter
	pSend:POINTER TO ARRAY[0..32767] OF BYTE; // Pointer to Send Buffer
	pSize:POINTER TO CAA.SIZE; // Send Size
END_VAR
VAR
	TransportHeader:SMB2_Transport_Header;
	SMB2Header: SMB2_Header_Sync;
	SMB2LogOff: SMB2_LOGOFF_Request;
	sendS:UINT;
	startIndex:UINT;
END_VAR

// This Function generates the LogOff Request

	// Increase Message ID
	Connection^.MessageID[0]:= Connection^.MessageID[0]+1;	
	// Create Header
	SMB2Header.ProtocolID[0]:= 16#FE; SMB2Header.ProtocolID[1]:= 16#53; SMB2Header.ProtocolID[2]:= 16#4D; SMB2Header.ProtocolID[3]:= 16#42; 
	SMB2Header.StructureSize := 64;
	SMB2Header.CreditCharge := 0;
	SMB2Header.Status := 0;
	SMB2Header.Command := Constants.LOGOFF;
	SMB2Header.CreditRepReq := 1;
	SMB2Header.Flags:= 0;
	SMB2Header.Flags := 0;
	SMB2Header.NextCommand := 0;		
	SMB2Header.MessageID[0]:= Connection^.MessageID[0]; SMB2Header.MessageID[1]:= 0;
	SMB2Header.TreeID:= 0;
	SMB2Header.SessionID[0]:= Connection^.Session.SessionID[0]; SMB2Header.SessionID[1]:= Connection^.Session.SessionID[1];
	SMB2Header.Signature[0]:= 0; SMB2Header.Signature[1]:= 0; SMB2Header.Signature[2]:= 0; SMB2Header.Signature[3]:= 0;
	
	// LogOff Request
	SMB2LogOff.StructureSize := 4;
	SMB2LogOff.Reserved := 0;
	
	// Copy Data in SendBuffer
	sendS:=SIZEOF(SMB2_Transport_Header);
	(*Parse SMB2 Header*)
	startIndex:=sendS-1;
	sendS:=sendS+SIZEOF(SMB2Header);
	MEM.MemMove(pSource:=ADR(SMB2Header) , pDestination:=ADR(pSend^[startIndex]) ,uiNumberOfBytes:=SIZEOF(SMB2Header));
	
	(*Parse LogOff Request*)
	startIndex:=sendS-1;
	sendS:=sendS+WORD_TO_UINT(SMB2LogOff.StructureSize);
	MEM.MemMove(pSource:=ADR(SMB2LogOff) , pDestination:=ADR(pSend^[startIndex]) ,uiNumberOfBytes:=WORD_TO_UINT(SMB2LogOff.StructureSize));
	
	(*Parse Transport Header*)
	TransportHeader.Zero := 16#00;
	TransportHeader.StreamProtocolLength := SHR(MEM.ReverseBYTEsInDWORD(sendS-SIZEOF(TransportHeader)),8);
		
	startIndex:=0;
	MEM.MemMove(pSource:=ADR(TransportHeader) , pDestination:=ADR(pSend^[startIndex]) ,uiNumberOfBytes:=SIZEOF(SMB2_Transport_Header)-1);
	
	(*Set Sendsize*)	
	pSize^:= sendS-1;

END_FUNCTION

// Device/Application/Bausteine/SMB2_Client/SMB2/Functions/Requests/CreateReq
FUNCTION CreateReq : int
VAR_INPUT
	Connection:POINTER TO Connection; // Connection Parameter
	pSend:POINTER TO ARRAY[0..32767] OF BYTE; // Pointer to Send Buffer
	pSize:POINTER TO CAA.SIZE; // Send Size
	fileName:WSTRING(256); // filename in SMB Server
	mode:INT; // 1= Send, 2= Receive, 3= Explorer (Dir/File Names), 4=srcsvc (Sharenames)
END_VAR
VAR
	i:INT;
	TransportHeader:SMB2_Transport_Header;
	SMB2Header: SMB2_Header_Sync;
	SMB2Create: SMB2_CREATE_Request;
	sendS:UINT;
	startIndex:UINT;
	pVar: POINTER TO ARRAY[0..255] OF BYTE;
	mode_3_length:WORD;
END_VAR

// This Function generates the Create Request

	// Increase Message ID
	Connection^.MessageID[0]:= Connection^.MessageID[0]+1;	
	// Create Header
	SMB2Header.ProtocolID[0]:= 16#FE; SMB2Header.ProtocolID[1]:= 16#53; SMB2Header.ProtocolID[2]:= 16#4D; SMB2Header.ProtocolID[3]:= 16#42; 
	SMB2Header.StructureSize := 64;
	SMB2Header.CreditCharge := 0;
	SMB2Header.Status := 0;
	SMB2Header.Command := Constants.CREATE;
	SMB2Header.CreditRepReq := 1;
	SMB2Header.Flags:= 0;
	SMB2Header.Flags := 0;
	SMB2Header.NextCommand := 0;		
	SMB2Header.MessageID[0]:= Connection^.MessageID[0]; SMB2Header.MessageID[1]:= 0;
	SMB2Header.TreeID:= connection^.Session.TreeConnect.TreeConnectId;
	SMB2Header.SessionID[0]:= Connection^.Session.SessionID[0]; SMB2Header.SessionID[1]:= Connection^.Session.SessionID[1];
	SMB2Header.Signature[0]:= 0; SMB2Header.Signature[1]:= 0; SMB2Header.Signature[2]:= 0; SMB2Header.Signature[3]:= 0;
	
	// Create Request
	SMB2Create.StructureSize:= 57;
	SMB2Create.SecurityFlags := 0;
	SMB2Create.RequestedOplockLevel := 16#08; // Named Pipe = 0
	SMB2Create.ImpersonationLevel := 2;
	SMB2Create.SmbCreateFlags[0] := 0; SMB2Create.SmbCreateFlags[1] := 0; // Must be 0
	SMB2Create.Reserved[0] := 0; SMB2Create.Reserved[1] := 0;
	IF mode = 1 THEN // Create new file or Open
		SMB2Create.DesiredAccess := 16#0017019F; // FILE_WRITE_DATA
		SMB2Create.FileAttributes := 16#00000020; // FILE_ATTRIBUTE_NORMAL
		SMB2Create.CreateDisposition := 16#00000005; // FILE_CREATE - If the file already exists, fail the operation; otherwise, create the file.
		SMB2Create.CreateOptions := 16#00000064;
		SMB2Create.ShareAccess := 0;	
	ELSIF mode = 2 THEN // Open File
		SMB2Create.DesiredAccess := 16#00100081; // 
		SMB2Create.FileAttributes := 16#00000000; // 
		SMB2Create.CreateDisposition := 16#00000001; // OPEN - if file exists open it, else fail
		SMB2Create.CreateOptions := 16#00000020;
		SMB2Create.ShareAccess := 16#00000007;	
	ELSIF mode = 3 THEN // Explorer
		SMB2Create.DesiredAccess := 16#00100081; // 
		SMB2Create.FileAttributes := 16#00000000; // 
		SMB2Create.CreateDisposition := 16#00000001; // OPEN - if file exists open it, else fail
		SMB2Create.CreateOptions := 16#00000020;
		SMB2Create.ShareAccess := 16#00000001;	
	ELSIF mode = 4 THEN // srvsvc
		SMB2Create.DesiredAccess := 16#0012019F; // 
		SMB2Create.FileAttributes := 16#00000000; // 
		SMB2Create.CreateDisposition := 16#00000001; // OPEN - if file exists open it, else fail
		SMB2Create.CreateOptions := 16#00000040;
		SMB2Create.ShareAccess := 16#00000007;	
	END_IF
	
	SMB2Create.NameOffset := 64+56;
	SMB2Create.NameLength := DINT_TO_WORD(wlen(fileName)*2);
	SMB2Create.CreateContextsLength := 0;
	SMB2Create.CreateContextsOffset := 0;
	pVar:=ADR(fileName);
	
	IF (WLEN(fileName) = 0) THEN // filename empty (explorer mode)
		SMB2Create.Payload[0]:= 0;
		SMB2Create.Payload[1]:= 0;
		mode_3_length:=2;
	ELSE
		FOR i:=0 TO WORD_TO_INT(SMB2Create.NameLength)-1 DO
		SMB2Create.Payload[i] := pVar^[i];
		mode_3_length:=0;
	END_FOR
		
	END_IF

	// Copy Data in SendBuffer
	sendS:=SIZEOF(SMB2_Transport_Header);
	(*Parse SMB2 Header*)
	startIndex:=sendS-1;
	sendS:=sendS+SIZEOF(SMB2Header);
	MEM.MemMove(pSource:=ADR(SMB2Header) , pDestination:=ADR(pSend^[startIndex]) ,uiNumberOfBytes:=SIZEOF(SMB2Header));
	
	(*Parse Create Request*)
	startIndex:=sendS-1;
	sendS:=sendS+WORD_TO_UINT(SMB2Create.StructureSize-1+SMB2Create.NameLength+mode_3_length);
	MEM.MemMove(pSource:=ADR(SMB2Create) , pDestination:=ADR(pSend^[startIndex]) ,uiNumberOfBytes:=WORD_TO_UINT(SMB2Create.StructureSize)-1+SMB2Create.NameLength+mode_3_length);
	
	(*Parse Transport Header*)
	TransportHeader.Zero := 16#00;
	TransportHeader.StreamProtocolLength := SHR(MEM.ReverseBYTEsInDWORD(sendS-SIZEOF(TransportHeader)),8);
		
	startIndex:=0;
	MEM.MemMove(pSource:=ADR(TransportHeader) , pDestination:=ADR(pSend^[startIndex]) ,uiNumberOfBytes:=SIZEOF(SMB2_Transport_Header)-1);
	
	(*Set Sendsize*)	
	pSize^:= sendS-1;

END_FUNCTION

// Device/Application/Bausteine/SMB2_Client/SMB2/Functions/Requests/QueryDirReq
FUNCTION QueryDirReq : int
VAR_INPUT
	Connection:POINTER TO Connection; // Connection Parameter
	pSend:POINTER TO ARRAY[0..32767] OF BYTE; // Pointer to Send Buffer
	pSize:POINTER TO CAA.SIZE; // Send Size
END_VAR
VAR
	i:INT;
	TransportHeader:SMB2_Transport_Header;
	SMB2Header: SMB2_Header_Sync;
	SMB2QueryDir: SMB2_QUERY_DIRECTORY_Request;
	sendS:UINT;
	startIndex:UINT;
	pVar: POINTER TO ARRAY[0..255] OF BYTE;
END_VAR

// This Function generates the Query Directory Request

	// Increase Message ID
	Connection^.MessageID[0]:= Connection^.MessageID[0]+1;	
	// Create Header
	SMB2Header.ProtocolID[0]:= 16#FE; SMB2Header.ProtocolID[1]:= 16#53; SMB2Header.ProtocolID[2]:= 16#4D; SMB2Header.ProtocolID[3]:= 16#42; 
	SMB2Header.StructureSize := 64;
	SMB2Header.CreditCharge := 0;
	SMB2Header.Status := 0;
	SMB2Header.Command := Constants.QUERY_DIRECTORY;
	SMB2Header.CreditRepReq := 1;
	SMB2Header.Flags:= 0;
	SMB2Header.Flags := 0;
	SMB2Header.NextCommand := 0;		
	SMB2Header.MessageID[0]:= Connection^.MessageID[0]; SMB2Header.MessageID[1]:= 0;
	SMB2Header.TreeID:= connection^.Session.TreeConnect.TreeConnectId;
	SMB2Header.SessionID[0]:= Connection^.Session.SessionID[0]; SMB2Header.SessionID[1]:= Connection^.Session.SessionID[1];
	SMB2Header.Signature[0]:= 0; SMB2Header.Signature[1]:= 0; SMB2Header.Signature[2]:= 0; SMB2Header.Signature[3]:= 0;
	
	// Query Directory Request
	SMB2QueryDir.StructureSize:= 33;
	SMB2QueryDir.FileInformationClass := 16#01; // Detailed information on the names of files and directories in a directory.
	SMB2QueryDir.Flags:= 0;
	SMB2QueryDir.FileIndex:=0;
	SMB2QueryDir.FileId:=Connection^.Session.Open.FileId;
	SMB2QueryDir.FileNameOffset:= 16#0060;
	SMB2QueryDir.FileNameLength:=2;
	SMB2QueryDir.OutputbufferLength:=8196;
	SMB2QueryDir.Payload[0]:= 16#2A; SMB2QueryDir.Payload[1]:= 16#00; // "*" für alles

	
	// Copy Data in SendBuffer
	sendS:=SIZEOF(SMB2_Transport_Header);
	(*Parse SMB2 Header*)
	startIndex:=sendS-1;
	sendS:=sendS+SIZEOF(SMB2Header);
	MEM.MemMove(pSource:=ADR(SMB2Header) , pDestination:=ADR(pSend^[startIndex]) ,uiNumberOfBytes:=SIZEOF(SMB2Header));
	
	(*Parse Query Directory Request*)
	startIndex:=sendS-1;
	sendS:=sendS+WORD_TO_UINT(SMB2QueryDir.StructureSize-1+SMB2QueryDir.FileNameLength);
	MEM.MemMove(pSource:=ADR(SMB2QueryDir) , pDestination:=ADR(pSend^[startIndex]) ,uiNumberOfBytes:=WORD_TO_UINT(SMB2QueryDir.StructureSize)-1+SMB2QueryDir.FileNameLength);
	
	(*Parse Transport Header*)
	TransportHeader.Zero := 16#00;
	TransportHeader.StreamProtocolLength := SHR(MEM.ReverseBYTEsInDWORD(sendS-SIZEOF(TransportHeader)),8);
		
	startIndex:=0;
	MEM.MemMove(pSource:=ADR(TransportHeader) , pDestination:=ADR(pSend^[startIndex]) ,uiNumberOfBytes:=SIZEOF(SMB2_Transport_Header)-1);
	
	(*Set Sendsize*)	
	pSize^:= sendS-1;

END_FUNCTION

// Device/Application/Bausteine/SMB2_Client/SMB2/Functions/NetShareBind
FUNCTION NetShareBind : int
VAR_INPUT
	Connection:POINTER TO Connection; // Connection Parameter
	pSend:POINTER TO ARRAY[0..32767] OF BYTE; // Pointer to Send Buffer
	pSize:POINTER TO CAA.SIZE; // Send Size
END_VAR
VAR
	i:INT;
	j:INT;
	TransportHeader:SMB2_Transport_Header;
	SMB2Header: SMB2_Header_Sync;
	SMB2Write: SMB2_WRITE_Request;
	sendS:UINT;
	startIndex:UINT;
	tempLWORD:LWORD;
	tempWORD:WORD;
	pVar: POINTER TO ARRAY[0..255] OF BYTE;
	tempwString:WSTRING;
	posFraglength:INT;
	posAllochint:INT;
	tempLenDRC:INT;
	srvsvcUID:ARRAY[0..15] OF BYTE:=[16#C8, 16#4F, 16#32, 16#4B, 16#70, 16#16, 16#D3, 16#01, 16#12, 16#78, 16#5A, 16#47, 16#BF, 16#6E, 16#E1, 16#88];
	ndrUID:ARRAY[0..15] OF BYTE:=[16#04, 16#5D, 16#88, 16#8A, 16#EB, 16#1C, 16#C9, 16#11, 16#9F, 16#E8, 16#08, 16#00, 16#2B, 16#10, 16#48, 16#60];
	ndrUIDV1:ARRAY[0..15] OF BYTE:=[16#33, 16#05, 16#71, 16#71, 16#BA, 16#BE, 16#37, 16#49, 16#83, 16#19, 16#B5, 16#DB, 16#EF, 16#9C, 16#CC, 16#36];
	bindUID:ARRAY[0..15] OF BYTE:=[16#2C, 16#1C, 16#B7, 16#6C, 16#12, 16#98, 16#40, 16#45, 16#03, 16#00, 16#00, 16#00, 16#00, 16#00, 16#00, 16#00];
END_VAR

// This function generates the NetShareBind, function is unknown, all Values and the Structure is copied from Wireshark

	// Increase Message ID
	Connection^.MessageID[0]:= Connection^.MessageID[0]+1;	
	// Create Header
	SMB2Header.ProtocolID[0]:= 16#FE; SMB2Header.ProtocolID[1]:= 16#53; SMB2Header.ProtocolID[2]:= 16#4D; SMB2Header.ProtocolID[3]:= 16#42; 
	SMB2Header.StructureSize := 64;
	SMB2Header.CreditCharge := 0;
	SMB2Header.Status := 0;
	SMB2Header.Command := Constants.write;
	SMB2Header.CreditRepReq := 1;
	SMB2Header.Flags:= 0;
	SMB2Header.Flags := 0;
	SMB2Header.NextCommand := 0;		
	SMB2Header.MessageID[0]:= Connection^.MessageID[0]; SMB2Header.MessageID[1]:= 0;
	SMB2Header.TreeID:= connection^.Session.TreeConnect.TreeConnectId;
	SMB2Header.SessionID[0]:= Connection^.Session.SessionID[0]; SMB2Header.SessionID[1]:= Connection^.Session.SessionID[1];
	SMB2Header.Signature[0]:= 0; SMB2Header.Signature[1]:= 0; SMB2Header.Signature[2]:= 0; SMB2Header.Signature[3]:= 0;
	
	// Write, all these values are copied from Wireshark
	SMB2Write.StructureSize:=16#0031;
	SMB2Write.DataOffset:=16#0070;
	SMB2Write.Length:=160;
	SMB2Write.Offset:=0;
	SMB2Write.FileId:= Connection[0].Session.Open.FileId;
	SMB2Write.Channel:=0;
	SMB2Write.WriteChannelInfoLength:=0;
	SMB2Write.RemainingBytes:=0;
	SMB2Write.Flags:=0;
	
	//Build DCE/RPC
	
	i:=16#70+4;
	
	pSend^[i]:=16#05; i:=i+1; // Version 5
	pSend^[i]:=16#00; i:=i+1; // Version Minor 0 -> 5.0
	pSend^[i]:=16#0B; i:=i+1; // Request Type (Bind)
	pSend^[i]:=16#03; i:=i+1; // Flags
	pSend^[i]:=16#10; i:=i+1; pSend^[i]:=16#00; i:=i+1; pSend^[i]:=16#00; i:=i+1; pSend^[i]:=16#00; i:=i+1; // Data Represantation (Little Endian, Char: ASCII, Float: IEEE)
	pSend^[i]:=16#A0; i:=i+1; pSend^[i]:=16#00; i:=i+1; // Frag Length
	pSend^[i]:=16#00; i:=i+1; pSend^[i]:=16#00; i:=i+1; // Auth Length
	pSend^[i]:=16#02; i:=i+1; pSend^[i]:=16#00; i:=i+1; pSend^[i]:=16#00; i:=i+1; pSend^[i]:=16#00; i:=i+1; // Call ID
	pSend^[i]:=16#B8; i:=i+1; pSend^[i]:=16#10; i:=i+1; // Max Xmit Frag
	pSend^[i]:=16#B8; i:=i+1; pSend^[i]:=16#10; i:=i+1; // Max Receive Frag
	pSend^[i]:=16#00; i:=i+1; pSend^[i]:=16#00; i:=i+1; pSend^[i]:=16#00; i:=i+1; pSend^[i]:=16#00; i:=i+1; // Asoc Group
	pSend^[i]:=16#03; i:=i+1; // Num Ctx Items - 3
	pSend^[i]:=16#00; i:=i+1; pSend^[i]:=16#00; i:=i+1; pSend^[i]:=16#00; i:=i+1; // Padding 3 bytes
	
	// Ctx Item 1
	pSend^[i]:=16#00; i:=i+1; pSend^[i]:=16#00; i:=i+1; // Context ID
	pSend^[i]:=16#01; i:=i+1; // Num Trans Items
	pSend^[i]:=16#00; i:=i+1; // Padding
	
	pVar:=ADR(srvsvcUID); // SRVSVC UID
	FOR j:=0 TO 15 DO
		pSend^[i]:= pVar^[j];
		i:=i+1;
	END_FOR
	pSend^[i]:=16#03; i:=i+1; pSend^[i]:=16#00; i:=i+1; // Interface Version 3
	pSend^[i]:=16#00; i:=i+1; pSend^[i]:=16#00; i:=i+1; // Version Minor 0 -> 3.0
	
	pVar:=ADR(ndrUID); // NDR UID
	FOR j:=0 TO 15 DO
		pSend^[i]:= pVar^[j];
		i:=i+1;
	END_FOR
	pSend^[i]:=16#02; i:=i+1; pSend^[i]:=16#00; i:=i+1; pSend^[i]:=16#00; i:=i+1; pSend^[i]:=16#00; i:=i+1; // Version 2
	
	// Ctx Item 2
	pSend^[i]:=16#01; i:=i+1; pSend^[i]:=16#00; i:=i+1; // Context ID 1
	pSend^[i]:=16#01; i:=i+1; // Num Trans Items
	pSend^[i]:=16#00; i:=i+1; // Padding
	
	pVar:=ADR(srvsvcUID); // SRVSVC UID
	FOR j:=0 TO 15 DO
		pSend^[i]:= pVar^[j];
		i:=i+1;
	END_FOR
	pSend^[i]:=16#03; i:=i+1; pSend^[i]:=16#00; i:=i+1; // Interface Version 3
	pSend^[i]:=16#00; i:=i+1; pSend^[i]:=16#00; i:=i+1; // Version Minor 0 -> 3.0
	
	pVar:=ADR(ndrUIDV1); // NDR UID
	FOR j:=0 TO 15 DO
		pSend^[i]:= pVar^[j];
		i:=i+1;
	END_FOR
	pSend^[i]:=16#01; i:=i+1; pSend^[i]:=16#00; i:=i+1; pSend^[i]:=16#00; i:=i+1; pSend^[i]:=16#00; i:=i+1; // Version 1
	
	// Ctx Item 3
	pSend^[i]:=16#02; i:=i+1; pSend^[i]:=16#00; i:=i+1; // Context ID 2
	pSend^[i]:=16#01; i:=i+1; // Num Trans Items
	pSend^[i]:=16#00; i:=i+1; // Padding
	
	pVar:=ADR(srvsvcUID); // SRVSVC UID
	FOR j:=0 TO 15 DO
		pSend^[i]:= pVar^[j];
		i:=i+1;
	END_FOR
	pSend^[i]:=16#03; i:=i+1; pSend^[i]:=16#00; i:=i+1; // Interface Version 3
	pSend^[i]:=16#00; i:=i+1; pSend^[i]:=16#00; i:=i+1; // Version Minor 0 -> 3.0
	
	pVar:=ADR(bindUID); // NDR UID
	FOR j:=0 TO 15 DO
		pSend^[i]:= pVar^[j];
		i:=i+1;
	END_FOR
	pSend^[i]:=16#01; i:=i+1; pSend^[i]:=16#00; i:=i+1; pSend^[i]:=16#00; i:=i+1; pSend^[i]:=16#00; i:=i+1; // Version 1
	
	// Copy Data in SendBuffer
	sendS:=SIZEOF(SMB2_Transport_Header);
	(*Parse SMB2 Header*)
	startIndex:=sendS-1;
	sendS:=sendS+SIZEOF(SMB2Header);
	MEM.MemMove(pSource:=ADR(SMB2Header) , pDestination:=ADR(pSend^[startIndex]) ,uiNumberOfBytes:=SIZEOF(SMB2Header));
	
	(*Parse IOCTL Request*)
	startIndex:=sendS-1;
	sendS:=sendS+WORD_TO_UINT(SMB2Write.StructureSize);
	MEM.MemMove(pSource:=ADR(SMB2Write) , pDestination:=ADR(pSend^[startIndex]) ,uiNumberOfBytes:=SIZEOF(SMB2Write));
	
	(*Parse Transport Header*)
	TransportHeader.Zero := 16#00;
	TransportHeader.StreamProtocolLength := SHR(MEM.ReverseBYTEsInDWORD(sendS+INT_TO_UINT(i-1-16#70-4)-SIZEOF(TransportHeader)),8);
		
	startIndex:=0;
	MEM.MemMove(pSource:=ADR(TransportHeader) , pDestination:=ADR(pSend^[startIndex]) ,uiNumberOfBytes:=SIZEOF(SMB2_Transport_Header)-1);
	
	(*Set Sendsize*)	
	pSize^:= sendS+INT_TO_UINT(i-1-16#70-4)-1;

END_FUNCTION

// Device/Application/Bausteine/SMB2_Client/SMB2/Functions/NetShareEnumAll
FUNCTION NetShareEnumAll : int
VAR_INPUT
	Connection:POINTER TO Connection; // Connection Parameter
	pSend:POINTER TO ARRAY[0..32767] OF BYTE; // Pointer to Send Buffer
	pSize:POINTER TO CAA.SIZE; // Send Size
END_VAR
VAR
	i:INT;
	j:INT;
	TransportHeader:SMB2_Transport_Header;
	SMB2Header: SMB2_Header_Sync;
	SMB2IO: SMB2_IOCTL_Request;
	sendS:UINT;
	startIndex:UINT;
	tempLWORD:LWORD;
	tempWORD:WORD;
	pVar: POINTER TO ARRAY[0..255] OF BYTE;
	tempwString:WSTRING;
	posFraglength:INT;
	posAllochint:INT;
	tempLenDRC:int;
END_VAR

// This function generates the NetShareEnumAll, all Values and the Structure is copied from Wireshark
// Response with all Share Names

	// Increase Message ID
	Connection^.MessageID[0]:= Connection^.MessageID[0]+1;	
	// Create Header
	SMB2Header.ProtocolID[0]:= 16#FE; SMB2Header.ProtocolID[1]:= 16#53; SMB2Header.ProtocolID[2]:= 16#4D; SMB2Header.ProtocolID[3]:= 16#42; 
	SMB2Header.StructureSize := 64;
	SMB2Header.CreditCharge := 0;
	SMB2Header.Status := 0;
	SMB2Header.Command := Constants.IOCTL;
	SMB2Header.CreditRepReq := 1;
	SMB2Header.Flags:= 0;
	SMB2Header.Flags := 0;
	SMB2Header.NextCommand := 0;		
	SMB2Header.MessageID[0]:= Connection^.MessageID[0]; SMB2Header.MessageID[1]:= 0;
	SMB2Header.TreeID:= connection^.Session.TreeConnect.TreeConnectId;
	SMB2Header.SessionID[0]:= Connection^.Session.SessionID[0]; SMB2Header.SessionID[1]:= Connection^.Session.SessionID[1];
	SMB2Header.Signature[0]:= 0; SMB2Header.Signature[1]:= 0; SMB2Header.Signature[2]:= 0; SMB2Header.Signature[3]:= 0;
	
	// IOCTL, all these values are copied from Wireshark
	SMB2IO.StructureSize:=16#0039;
	SMB2IO.Reserved:=0;
	SMB2IO.CtlCode:=16#0011C017;
	SMB2IO.FileID:=Connection[0].Session.Open.FileId;
	SMB2IO.InputOffset:=16#00000078;
	SMB2IO.MaxInputResponse:=0;
	SMB2IO.OutputOffset:=16#00000078;
	SMB2IO.OutputCount:=0;
	SMB2IO.MaxOutputResponse:=8192;
	SMB2IO.Flags:=16#00000001;
	SMB2IO.Reserved2:=0;
	
	//Build DCE/RPC
	
	i:=16#78+4;
	
	pSend^[i]:=16#05; i:=i+1; // Version 5
	pSend^[i]:=16#00; i:=i+1; // Version Minor 0 -> 5.0
	pSend^[i]:=16#00; i:=i+1; // Request Type
	pSend^[i]:=16#03; i:=i+1; // Flags
	pSend^[i]:=16#10; i:=i+1; pSend^[i]:=16#00; i:=i+1; pSend^[i]:=16#00; i:=i+1; pSend^[i]:=16#00; i:=i+1; // Data Represantation (Little Endian, Char: ASCII, Float: IEEE)
	posFraglength:=i; i:=i+2;// Frag Length, Save Position
	pSend^[i]:=16#00; i:=i+1; pSend^[i]:=16#00; i:=i+1; // Auth Length
	pSend^[i]:=16#02; i:=i+1; pSend^[i]:=16#00; i:=i+1; pSend^[i]:=16#00; i:=i+1; pSend^[i]:=16#00; i:=i+1; // Call ID
	posAllocHint:=i; i:=i+4; // Alloc Hint <-- Length of Netshareenum, Save Position
	pSend^[i]:=16#01; i:=i+1; pSend^[i]:=16#00; i:=i+1; // Context ID ?
	pSend^[i]:=16#0F; i:=i+1; pSend^[i]:=16#00; i:=i+1; // OpNum = NetShareEnumAll
	
	tempLenDRC:=i-16#78-4; // Save Length of DRC for Alloc Hint
	
	// Build NetShareEnumAll
	// Pointer to Server Unc
	tempLWORD:= 16#0000000000020000; pVar:=ADR(tempLWORD); // Referant ID
	FOR j:=0 TO 7 DO
		pSend^[i]:= pVar^[j];
		i:=i+1;
	END_FOR
	
	tempwString := wconcat("\\",Connection^.wServerName);
	tempLWORD:= INT_TO_LWORD(wlen(tempwString))+1; pVar:=ADR(tempLWORD); // Length Servername
	FOR j:=0 TO 7 DO
		pSend^[i]:= pVar^[j];
		i:=i+1;
	END_FOR
	
	tempLWORD:= 0; pVar:=ADR(tempLWORD); // Offset
	FOR j:=0 TO 7 DO
		pSend^[i]:= pVar^[j];
		i:=i+1;
	END_FOR
	
	tempLWORD:= INT_TO_LWORD(wlen(tempwString))+1; pVar:=ADR(tempLWORD); // Acutal Count
	FOR j:=0 TO 7 DO
		pSend^[i]:= pVar^[j];
		i:=i+1;
	END_FOR
	
	// Server UNC
	pVar:=ADR(tempwString); // Server Name
	FOR j:=0 TO wlen(tempwString)*2+1 DO
		pSend^[i]:= pVar^[j];
		i:=i+1;
	END_FOR
	
	IF (((WLEN(tempwString)+1)*2) MOD 8) > 0 THEN // padding after name
		FOR j:=0 TO 8-(((WLEN(tempwString)+1)*2) MOD 8)-1 DO
			pSend^[i]:= 16#00;
			i:=i+1;
		END_FOR
	END_IF
	pSend^[i]:=16#01; i:=i+1; pSend^[i]:=16#00; i:=i+1; pSend^[i]:=16#00; i:=i+1; pSend^[i]:=16#00; i:=i+1; // Pointer to Level
	// Pointer to Ctr
	pSend^[i]:=16#00; i:=i+1; pSend^[i]:=16#00; i:=i+1; pSend^[i]:=16#00; i:=i+1; pSend^[i]:=16#00; i:=i+1; // Ctr
	// Pointer to Ctr0
	tempLWORD:= 16#0000000000000001; pVar:=ADR(tempLWORD); // Referant ID
	FOR j:=0 TO 7 DO
		pSend^[i]:= pVar^[j];
		i:=i+1;
	END_FOR
	// Ctr0
	pSend^[i]:=16#00; i:=i+1; pSend^[i]:=16#00; i:=i+1; pSend^[i]:=16#02; i:=i+1; pSend^[i]:=16#00; i:=i+1; // Count ?
	pSend^[i]:=16#00; i:=i+1; pSend^[i]:=16#00; i:=i+1; pSend^[i]:=16#00; i:=i+1; pSend^[i]:=16#00; i:=i+1; // Reserved?
	tempLWORD:= 16#00; pVar:=ADR(tempLWORD); // NULL Pointer
	FOR j:=0 TO 7 DO
		pSend^[i]:= pVar^[j];
		i:=i+1;
	END_FOR
	pSend^[i]:=16#00; i:=i+1; pSend^[i]:=16#00; i:=i+1; pSend^[i]:=16#00; i:=i+1; pSend^[i]:=16#00; i:=i+1; // Max Buffer
	pSend^[i]:=16#00; i:=i+1; pSend^[i]:=16#00; i:=i+1; pSend^[i]:=16#00; i:=i+1; pSend^[i]:=16#00; i:=i+1; // Reserved?
	// Pointer to Resume Handle
	tempLWORD:= 16#00000000FFFFFFFF; pVar:=ADR(tempLWORD); // Referant ID
	FOR j:=0 TO 7 DO
		pSend^[i]:= pVar^[j];
		i:=i+1;
	END_FOR
	pSend^[i]:=16#00; i:=i+1; pSend^[i]:=16#00; i:=i+1; pSend^[i]:=16#00; i:=i+1; pSend^[i]:=16#00; i:=i+1; // Resume Handle
	pSend^[i]:=16#00; i:=i+1; pSend^[i]:=16#00; i:=i+1; pSend^[i]:=16#00; i:=i+1; pSend^[i]:=16#00; i:=i+1; // Long Frame
	
	// Insert Length at the End
	tempWORD:= INT_TO_WORD(i-16#78-4);  pVar:=ADR(tempWORD); // Frag Length
	FOR j:=0 TO 1 DO
		pSend^[j+posFraglength]:= pVar^[j];
	END_FOR
	
	tempLWORD:= INT_TO_LWORD(i-16#78-4-tempLenDRC);  pVar:=ADR(tempLWORD); // Alloc Hint
	FOR j:=0 TO 3 DO
		pSend^[j+posAllocHint]:= pVar^[j];
	END_FOR
	
	SMB2IO.InputCount:= INT_TO_DWORD(i-16#78-4);
	

	// Copy Data in SendBuffer
	sendS:=SIZEOF(SMB2_Transport_Header);
	(*Parse SMB2 Header*)
	startIndex:=sendS-1;
	sendS:=sendS+SIZEOF(SMB2Header);
	MEM.MemMove(pSource:=ADR(SMB2Header) , pDestination:=ADR(pSend^[startIndex]) ,uiNumberOfBytes:=SIZEOF(SMB2Header));
	
	(*Parse IOCTL Request*)
	startIndex:=sendS-1;
	sendS:=sendS+WORD_TO_UINT(SMB2IO.StructureSize);
	MEM.MemMove(pSource:=ADR(SMB2IO) , pDestination:=ADR(pSend^[startIndex]) ,uiNumberOfBytes:=SIZEOF(SMB2IO));
	
	(*Parse Transport Header*)
	TransportHeader.Zero := 16#00;
	TransportHeader.StreamProtocolLength := SHR(MEM.ReverseBYTEsInDWORD(sendS+INT_TO_UINT(i-1-16#78-4)-SIZEOF(TransportHeader)),8);
		
	startIndex:=0;
	MEM.MemMove(pSource:=ADR(TransportHeader) , pDestination:=ADR(pSend^[startIndex]) ,uiNumberOfBytes:=SIZEOF(SMB2_Transport_Header)-1);
	
	(*Set Sendsize*)	
	pSize^:= sendS+INT_TO_UINT(i-1-16#78-4)-1;

END_FUNCTION

// Device/Application/Bausteine/SMB2_Client/SMB2/Functions/Requests/ReadRequest
FUNCTION ReadRequest : INT
VAR_INPUT
	Connection:POINTER TO Connection; // Connection Parameter
	pSend:POINTER TO ARRAY[0..32767] OF BYTE; // Pointer to Send Buffer
	pSize:POINTER TO CAA.SIZE;  // Send Size
	numBytes:UINT; // number of bytes to read
END_VAR
VAR
	TransportHeader:SMB2_Transport_Header;
	SMB2Header: SMB2_Header_Sync;
	SMB2Read:SMB2_READ_Request;
	
	sendS:UINT;
	startIndex:UINT;
	i:INT;
END_VAR

// This Function generates the Read Request Request

		// Increase Message ID
		Connection^.MessageID[0]:= Connection^.MessageID[0]+1;	
		// Create Header
		SMB2Header.ProtocolID[0]:= 16#FE; SMB2Header.ProtocolID[1]:= 16#53; SMB2Header.ProtocolID[2]:= 16#4D; SMB2Header.ProtocolID[3]:= 16#42; 
		SMB2Header.StructureSize := 64;
		SMB2Header.CreditCharge := 0;
		SMB2Header.Status := 0;
		SMB2Header.Command := Constants.READ;
		SMB2Header.CreditRepReq := 0;
		SMB2Header.Flags:= 0;
		SMB2Header.Flags := 0;
		SMB2Header.NextCommand := 0;		
		SMB2Header.MessageID[0]:= Connection^.MessageID[0]; SMB2Header.MessageID[1]:= 0;
		SMB2Header.Reserved := 0;
		SMB2Header.TreeID:= connection^.Session.TreeConnect.TreeConnectId;
		SMB2Header.SessionID[0]:= Connection^.Session.SessionID[0];; SMB2Header.SessionID[1]:= Connection^.Session.SessionID[1];
		SMB2Header.Signature[0]:= 0; SMB2Header.Signature[1]:= 0; SMB2Header.Signature[2]:= 0; SMB2Header.Signature[3]:= 0;
			
		// Read Message Request
		SMB2Read.Padding:= 16#50;
		SMB2Read.Length := numBytes;
		SMB2Read.Offset:= 0;
		SMB2Read.FileId:= Connection[0].Session.Open.FileId;
		
		// Copy Data in SendBuffer
		sendS:=SIZEOF(SMB2_Transport_Header);
		(*Parse SMB2 Header*)
		startIndex:=sendS-1;
		sendS:=sendS+SIZEOF(SMB2Header);
		MEM.MemMove(pSource:=ADR(SMB2Header) , pDestination:=ADR(pSend^[startIndex]) ,uiNumberOfBytes:=SIZEOF(SMB2Header));
		
		(*Parse Read Request*)
		startIndex:=sendS-1;
		sendS:=sendS+1+WORD_TO_UINT(SMB2Read.StructureSize-1);
		MEM.MemMove(pSource:=ADR(SMB2Read) , pDestination:=ADR(pSend^[startIndex]) ,uiNumberOfBytes:=WORD_TO_UINT(SMB2Read.StructureSize)-1);
				
		(*Parse Transport Header*)
		TransportHeader.Zero := 16#00;
		TransportHeader.StreamProtocolLength := SHR(MEM.ReverseBYTEsInDWORD(sendS-SIZEOF(TransportHeader)),8);
				
		startIndex:=0;
		MEM.MemMove(pSource:=ADR(TransportHeader) , pDestination:=ADR(pSend^[startIndex]) ,uiNumberOfBytes:=SIZEOF(SMB2_Transport_Header)-1);
			
		(*Set Sendsize*)	
		pSize^:= sendS-1;

END_FUNCTION

// Device/Application/Bausteine/SMB2_Client/SMB2/Functions/SendFile
FUNCTION_BLOCK SendFile
VAR_INPUT
	xExecute:BOOL; // Start Routine
	Connection:POINTER TO Connection; // Connection Parameter
	pSend:POINTER TO ARRAY[0..65536] OF BYTE; // Pointer to Send Buffer
	pSize:POINTER TO CAA.SIZE; // Send Size
	filePath:STRING; // Filepath on PLC
	bufferSize:UDINT; // Send/Receive Buffer Size
	nextRound:BOOL; // Ready for next round
END_VAR
VAR_OUTPUT
	xDone:BOOL;
	send:BOOL;
	xError:BOOL;
END_VAR
VAR
	step:INT:=1;
	getSize:FILE.GetSize;
	open:FILE.Open;
	close:File.Close;
	read:file.Read;
	fileSize:UDINT;
	remaining:UDINT;
	TransportHeader:SMB2_Transport_Header;
	SMB2Header: SMB2_Header_Sync;
	SMB2Write:SMB2_WRITE_Request;
	sendS:UINT;
	startIndex:UINT;
	i:INT;
	roundsMax:UDINT;
	roundsAct:UDINT;
	SMB2WriteFileId: INT;
	hFile:CAA.HANDLE;
END_VAR

// This FB sends Files from SD-Card to SMB Server


IF NOT xExecute THEN
	step:=0;
END_IF
xDone := FALSE;
xError:= FALSE;
CASE step OF
	
	0:	step:=step+1;
		send:=FALSE;
		// Get Size of File on PLC
	1: 	getSize.xExecute:=TRUE;
		IF getSize.xDone THEN
			fileSize := getSize.szSize;
			roundsAct:= 1;
			roundsMax:= (fileSize/bufferSize) + 1; // Number of Round, Buffer smaller than size of file
			getSize.xExecute:=FALSE;
			step:=step+1;
		END_IF
		
	2:	// Open File, get file handle on PLC
	   open.xExecute := TRUE;
        IF open.xDone THEN
			open.xExecute := FALSE;
            hFile:=open.hFile;
            step:=step+1;
        END_IF
	
		// Create or Open File on Server (Create Request)
	3: 	CreateReq(Connection:=Connection,pSend:=pSend,pSize:=pSize,fileName:=Connection^.requestedFileName,mode:=1);
		send:=TRUE;
		step:=step+1;
	4:	IF nextRound THEN
			send:=FALSE;
			step:=step+1;
		END_IF

	5:	// Build Write Message
		// Increase Message ID
		Connection^.MessageID[0]:= Connection^.MessageID[0]+1;	
		// Create Header
		SMB2Header.ProtocolID[0]:= 16#FE; SMB2Header.ProtocolID[1]:= 16#53; SMB2Header.ProtocolID[2]:= 16#4D; SMB2Header.ProtocolID[3]:= 16#42; 
		SMB2Header.StructureSize := 64;
		SMB2Header.CreditCharge := 0;
		SMB2Header.Status := 0;
		SMB2Header.Command := Constants.WRITE;
		SMB2Header.CreditRepReq := 111;
		SMB2Header.Flags:= 0;
		SMB2Header.Flags := 0;
		SMB2Header.NextCommand := 0;		
		SMB2Header.MessageID[0]:= Connection^.MessageID[0]; SMB2Header.MessageID[1]:= 0;
		SMB2Header.TreeID:= connection^.Session.TreeConnect.TreeConnectId;
		SMB2Header.SessionID[0]:= Connection^.Session.SessionID[0]; SMB2Header.SessionID[1]:= Connection^.Session.SessionID[1];
		SMB2Header.Signature[0]:= 0; SMB2Header.Signature[1]:= 0; SMB2Header.Signature[2]:= 0; SMB2Header.Signature[3]:= 0;
				
		step:=step+1;
			
	6:	// Write Message Request
		SMB2Write.DataOffset:= 64+48;
		IF roundsAct = roundsMax THEN
			SMB2Write.Length := UDINT_TO_DWORD(fileSize - (roundsAct-1)*bufferSize); // write remaining bytes to read length
		ELSE
			SMB2Write.Length := UDINT_TO_DWORD(bufferSize); // write buffersize to read length
		END_IF
		SMB2Write.Offset:= LINT_TO_LWORD((roundsAct-1)*UDINT_TO_LINT(bufferSize)); // Fileoffset on Server
		SMB2Write.FileId:= Connection[0].Session.Open.FileId; // File ID of opened file on Server
		SMB2Write.RemainingBytes:= UDINT_TO_WORD(fileSize - DWORD_TO_UDINT(SMB2Write.Length) - (roundsAct-1)*bufferSize); // Remaining bytes to send after this operation
		
		// Copy Data in SendBuffer
		sendS:=SIZEOF(SMB2_Transport_Header);
		(*Parse SMB2 Header*)
		startIndex:=sendS-1;
		sendS:=sendS+SIZEOF(SMB2Header);
		MEM.MemMove(pSource:=ADR(SMB2Header) , pDestination:=ADR(pSend^[startIndex]) ,uiNumberOfBytes:=SIZEOF(SMB2Header));
		
		(*Parse Write Request*)
		startIndex:=sendS-1;
		sendS:=sendS+WORD_TO_UINT(SMB2Write.StructureSize-1);
		MEM.MemMove(pSource:=ADR(SMB2Write) , pDestination:=ADR(pSend^[startIndex]) ,uiNumberOfBytes:=WORD_TO_UINT(SMB2Write.StructureSize)-1);
				
		step:=step+1;
		
	7: 	(*Parse Payload*)
		startIndex:=sendS-1;
		sendS:= sendS + DWORD_TO_UINT(SMB2Write.Length);
		
		step:=step+1;
		
    8:	// Copy bytes from file into send buffer - after that calcualte length of Message and send to Server
		read.xExecute:= TRUE;
		IF read.xDone THEN
			read.xExecute:= FALSE;
			
			(*Parse Transport Header*)
			TransportHeader.Zero := 16#00;
			TransportHeader.StreamProtocolLength := SHR(MEM.ReverseBYTEsInDWORD(sendS-SIZEOF(TransportHeader)),8);
				
			startIndex:=0;
			MEM.MemMove(pSource:=ADR(TransportHeader) , pDestination:=ADR(pSend^[startIndex]) ,uiNumberOfBytes:=SIZEOF(SMB2_Transport_Header)-1);
			
			(*Set Sendsize*)	
			pSize^:= sendS-1;
			send:=TRUE;
			
            step:=step+1;
        END_IF

	9:	// send ready (nextround)
		IF nextRound THEN
			send:=FALSE;
			IF roundsAct = roundsMax THEN // all bytes send
				step:=step+1;
			ELSE			// next round
				step:=5;		
			END_IF	
			roundsAct:=roundsAct+1;
		END_IF
		
	10: // Close File on PLC
		close.xExecute:= TRUE;
		IF close.xDone THEN
			close.xExecute:= FALSE;
			step:=1;
			xDone:=TRUE;
		END_IF

END_CASE

// Error
IF open.xError OR read.xError OR close.xError THEN
	xError := TRUE;
	step:=1;
END_IF

// Open, Read, Close File on PLC - Must be called every cycle
getSize(sFileName:=filePath);
open(xExclusive:=TRUE,eFileMode:=FILE.MODE.MREAD,sFileName:=filePath); // Opens a file on the PLC
read(hFile:=hFile,pBuffer:=ADR(pSend^[startIndex]),szBuffer:=bufferSize, udiTimeOut:=100000); // read from file into send buffer
close(hFile:=hFile); // Close file on PLC

END_FUNCTION_BLOCK

// Device/Application/Bausteine/SMB2_Client/SMB2/Functions/ReadFile
FUNCTION_BLOCK ReadFile
VAR_INPUT
	xExecute:BOOL; // Start Routine
	Connection:POINTER TO Connection; // Connection Parameter
	pSend:POINTER TO ARRAY[0..65536] OF BYTE; // Pointer to Send Buffer
	pSize:POINTER TO CAA.SIZE; // Send Size
	pRecv:POINTER TO ARRAY[0..65536] OF BYTE; // Pointer to Receive Buffer
	filePath:STRING; // Filepath on PLC
	bufferSize:UDINT; // Send/Receive Buffer Size
	nextRound:BOOL; // Ready for next round
	received:BOOL; // New Data in Receive Buffer
END_VAR
VAR_OUTPUT
	xDone:BOOL;
	send:BOOL;
	xError:BOOL;
END_VAR
VAR
	step:INT:=1;
	fileSize:ARRAY[0..1] OF UDINT;
	
	open:FILE.Open;
	close:File.Close;
	write:File.Write;
	hFile:CAA.HANDLE;


	

	remaining:UDINT;
	TransportHeader:SMB2_Transport_Header;
	SMB2Header: SMB2_Header_Sync;
	SMB2Read:SMB2_READ_Request;
	
	sendS:UINT;
	startIndex:UINT;
	i:INT;
	roundsMax:UDINT;
	roundsAct:UDINT;
	SMB2WriteFileId: INT;
END_VAR

// This FB read files from SMB Server to SD-Card

IF NOT xExecute THEN
	step:=0;
END_IF
xDone := FALSE;
xError:= FALSE;
CASE step OF
	
	0: 	step:=step+1;
		// Create File / Open File on Server (Create Request)
	1: 	CreateReq(Connection:=Connection,pSend:=pSend,pSize:=pSize,fileName:=Connection^.requestedFileName, Mode:=2); // Create Request, Open File with Filename on Server
		send:=TRUE;
		step:=step+1;
		
	2:	IF received THEN // Create Request sucessful
			send:=FALSE;
			fileSize[0] := Connection^.Session.Open.FileSize[0]; fileSize[1] := Connection^.Session.Open.FileSize[1]; // File Size on PC (End of File)
			step:=step+1;
		END_IF
		
	3: // Create File on PLC
		open.xExecute:=TRUE; // Open File on SD-Card
		roundsAct:= 1; // Actual number of rounds
		roundsMax:= (fileSize[0]/bufferSize) + 1; // Number of Rounds, because Buffer smaller than size of file
        IF open.xDone THEN // File on SD-Card opened
			open.xExecute:=FALSE;
            hFile:=open.hFile; // File Handle
            step:=step+1;
        END_IF
		
	4:	// Build SMB2 Header and Readrequest
		// Increase Message ID
		Connection^.MessageID[0]:= Connection^.MessageID[0]+1;	
		// Create Header
		SMB2Header.ProtocolID[0]:= 16#FE; SMB2Header.ProtocolID[1]:= 16#53; SMB2Header.ProtocolID[2]:= 16#4D; SMB2Header.ProtocolID[3]:= 16#42; 
		SMB2Header.StructureSize := 64;
		SMB2Header.CreditCharge := 0;
		SMB2Header.Status := 0;
		SMB2Header.Command := Constants.READ;
		SMB2Header.CreditRepReq := 0;
		SMB2Header.Flags:= 0;
		SMB2Header.Flags := 0;
		SMB2Header.NextCommand := 0;		
		SMB2Header.MessageID[0]:= Connection^.MessageID[0]; SMB2Header.MessageID[1]:= 0;
		SMB2Header.Reserved := 0;
		SMB2Header.TreeID:= connection^.Session.TreeConnect.TreeConnectId;
		SMB2Header.SessionID[0]:= Connection^.Session.SessionID[0];; SMB2Header.SessionID[1]:= Connection^.Session.SessionID[1];
		SMB2Header.Signature[0]:= 0; SMB2Header.Signature[1]:= 0; SMB2Header.Signature[2]:= 0; SMB2Header.Signature[3]:= 0;
		
		
		step:=step+1;
		
		
	5:	// Read Message Request
		SMB2Read.Padding:= 16#50;
		IF roundsAct = roundsMax THEN // Last round
			SMB2Read.Length := UDINT_TO_DWORD(fileSize[0] - (roundsAct-1)*bufferSize); // write remaining bytes to read length in request 
		ELSE
			SMB2Read.Length := UDINT_TO_DWORD(bufferSize); // write buffersize to read length, read max buffersize
		END_IF
		SMB2Read.Offset:= ULINT_TO_LWORD((roundsAct-1)*UDINT_TO_ULINT(bufferSize)); // Fileoffset on Server
		SMB2Read.FileId:= Connection[0].Session.Open.FileId; // File ID of opened file on Server
		
		// Copy Data in SendBuffer
		sendS:=SIZEOF(SMB2_Transport_Header);
		(*Parse SMB2 Header*)
		startIndex:=sendS-1;
		sendS:=sendS+SIZEOF(SMB2Header);
		MEM.MemMove(pSource:=ADR(SMB2Header) , pDestination:=ADR(pSend^[startIndex]) ,uiNumberOfBytes:=SIZEOF(SMB2Header));
		
		(*Parse Write Request*)
		startIndex:=sendS-1;
		sendS:=sendS+1+WORD_TO_UINT(SMB2Read.StructureSize-1);
		MEM.MemMove(pSource:=ADR(SMB2Read) , pDestination:=ADR(pSend^[startIndex]) ,uiNumberOfBytes:=WORD_TO_UINT(SMB2Read.StructureSize)-1);
				
		(*Parse Transport Header*)
		TransportHeader.Zero := 16#00;
		TransportHeader.StreamProtocolLength := SHR(MEM.ReverseBYTEsInDWORD(sendS-SIZEOF(TransportHeader)),8);
				
		startIndex:=0;
		MEM.MemMove(pSource:=ADR(TransportHeader) , pDestination:=ADR(pSend^[startIndex]) ,uiNumberOfBytes:=SIZEOF(SMB2_Transport_Header)-1);
			
		(*Set Sendsize*)	
		pSize^:= sendS-1;
		send:=TRUE;
			
		step:=step+1;
		
	6:	IF received THEN // Read Request sucessful
			send:=FALSE;
			step:=step+1;
		END_IF
		
	7: // Write Buffer to Disk
		write.xExecute:= TRUE; // Start write Read Response Data to SD-Card
 		IF write.xDone THEN // Write sucessful
			write.xExecute:= FALSE;
			IF roundsAct = roundsMax THEN // all bytes send
				step:=8;
			ELSE				// next round
				step:=4;		
			END_IF	
			roundsAct:=roundsAct+1;
		END_IF
		
	8:	// Close File on PLC
		close.xExecute:=TRUE; // Close file on SD-Card
		IF close.xDone THEN
			close.xExecute:=FALSE;
			step:=1;
			xDone:=TRUE;
		END_IF

END_CASE

// Error
IF open.xError OR write.xError OR close.xError THEN
	xError := TRUE;
	step:=1;
END_IF

// Open, Write, Close File on PLC - Must be called every cycle
open(xExclusive:=TRUE,eFileMode:=FILE.MODE.MWRITE,sFileName:=filePath); // Opens a file on the PLC
write(hFile:=hFile,pBuffer:=ADR(pRecv^[Connection^.Session.Open.ReadDataOffset+4]),szSize:=Connection^.Session.Open.ReadDataLength, udiTimeOut:=1000000); // write send buffer to disk
close(hFile:=hFile); // Close file on PLC

END_FUNCTION_BLOCK

// Device/Application/Start
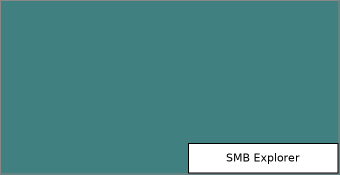
VISUALIZATION Start  // 340x175
    Rectangle (188,143 150x30), "SMB Explorer"
        OnMouseUp:  Assign=SMB_Explorer, Type=Assignment
END_VISUALIZATION

// Device/Application/SMB_Explorer
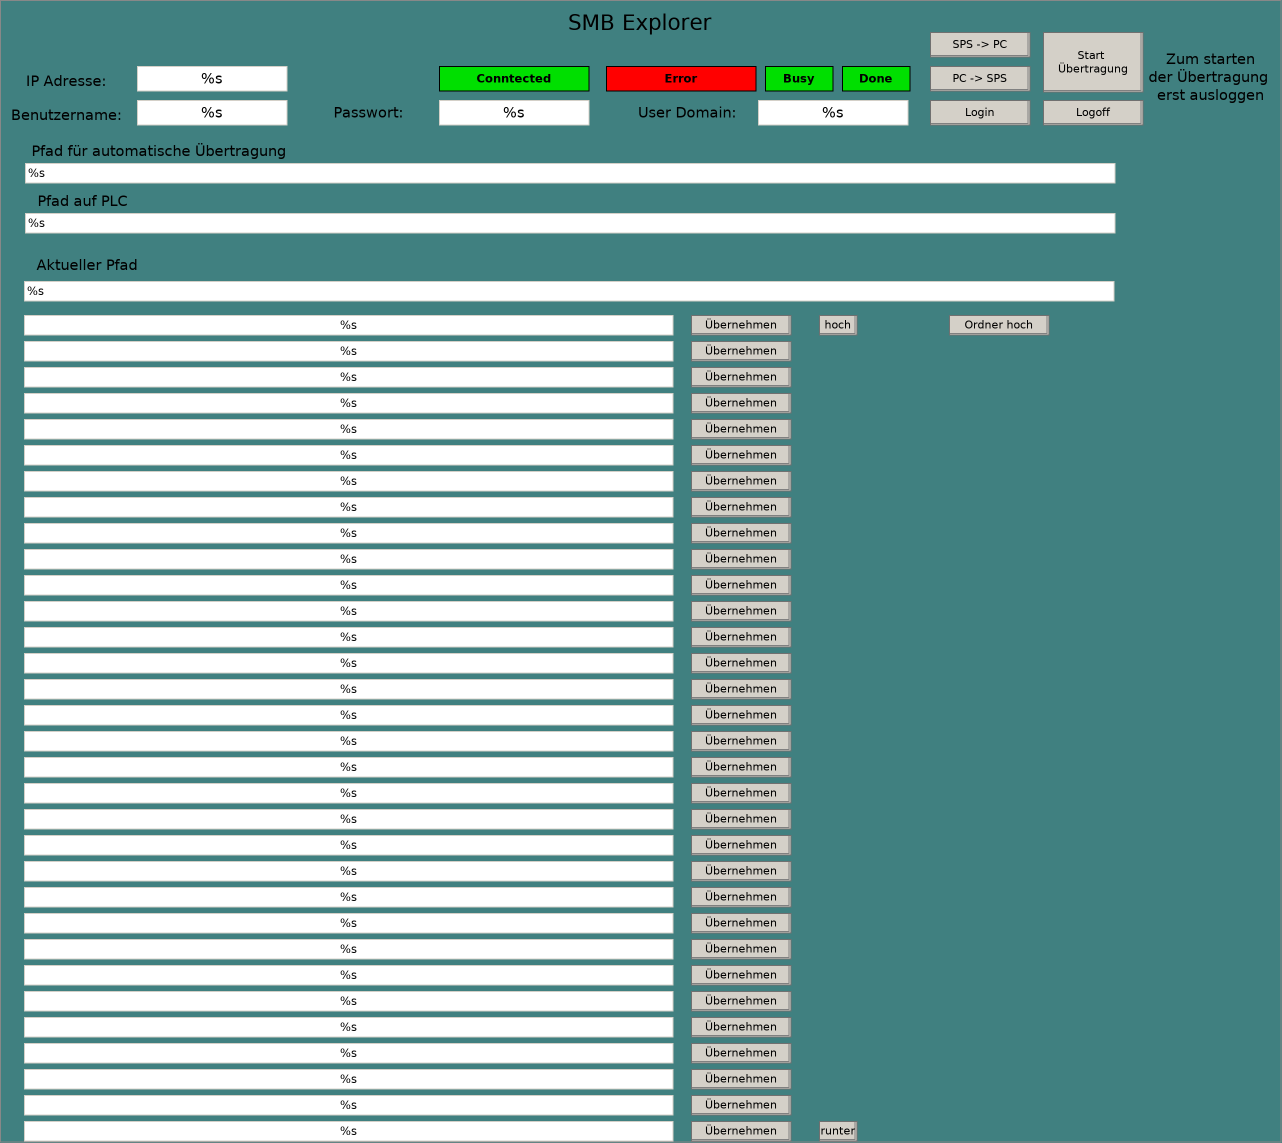
VISUALIZATION SMB_Explorer  // 1282x1143
    Textfield (137,100 150x25), "%s", text variable: VAR_Explorer.Visu_Explorer.User
        OnMouseDown: write the text variable via Edit
    Label (0,0 1280x45), "SMB Explorer"
    Label (1,100 131x30), "Benutzername:"
    Textfield (439,100 150x25), "%s", text variable: VAR_Explorer.Visu_Explorer.Password
        OnMouseDown: write the text variable via Edit
    Label (303,100 131x25), "Passwort:"
    Textfield (758,100 150x25), "%s", text variable: VAR_Explorer.Visu_Explorer.UserDomain
        OnMouseDown: write the text variable via Edit
    Label (622,100 131x25), "User Domain:"
    Textfield (137,66 150x25), "%s", text variable: VAR_Explorer.Visu_Explorer.IPAdress
        OnMouseDown: write the text variable via Edit
    Label (1,66 131x30), "IP Adresse:"
    Textfield (24,315 649x20), "%s", text variable: VAR_Explorer.Visu_Explorer.Directory[VAR_Explorer.Visu_Explorer.DirectoryIndex+0]
    Button (930,100 100x25), "Login"
        tap VAR_Explorer.Visu_Explorer.Login
    Button (1043,100 100x25), "Logoff"
        tap VAR_Explorer.Visu_Explorer.Logout
    Textfield (24,341 649x20), "%s", text variable: VAR_Explorer.Visu_Explorer.Directory[VAR_Explorer.Visu_Explorer.DirectoryIndex+1]
    Textfield (24,367 649x20), "%s", text variable: VAR_Explorer.Visu_Explorer.Directory[VAR_Explorer.Visu_Explorer.DirectoryIndex+2]
    Textfield (24,393 649x20), "%s", text variable: VAR_Explorer.Visu_Explorer.Directory[VAR_Explorer.Visu_Explorer.DirectoryIndex+3]
    Textfield (24,419 649x20), "%s", text variable: VAR_Explorer.Visu_Explorer.Directory[VAR_Explorer.Visu_Explorer.DirectoryIndex+4]
    Textfield (24,445 649x20), "%s", text variable: VAR_Explorer.Visu_Explorer.Directory[VAR_Explorer.Visu_Explorer.DirectoryIndex+5]
    Textfield (24,471 649x20), "%s", text variable: VAR_Explorer.Visu_Explorer.Directory[VAR_Explorer.Visu_Explorer.DirectoryIndex+6]
    Textfield (24,497 649x20), "%s", text variable: VAR_Explorer.Visu_Explorer.Directory[VAR_Explorer.Visu_Explorer.DirectoryIndex+7]
    Textfield (24,523 649x20), "%s", text variable: VAR_Explorer.Visu_Explorer.Directory[VAR_Explorer.Visu_Explorer.DirectoryIndex+8]
    Textfield (24,549 649x20), "%s", text variable: VAR_Explorer.Visu_Explorer.Directory[VAR_Explorer.Visu_Explorer.DirectoryIndex+9]
    Textfield (24,575 649x20), "%s", text variable: VAR_Explorer.Visu_Explorer.Directory[VAR_Explorer.Visu_Explorer.DirectoryIndex+10]
    Textfield (24,601 649x20), "%s", text variable: VAR_Explorer.Visu_Explorer.Directory[VAR_Explorer.Visu_Explorer.DirectoryIndex+11]
    Textfield (24,627 649x20), "%s", text variable: VAR_Explorer.Visu_Explorer.Directory[VAR_Explorer.Visu_Explorer.DirectoryIndex+12]
    Textfield (24,653 649x20), "%s", text variable: VAR_Explorer.Visu_Explorer.Directory[VAR_Explorer.Visu_Explorer.DirectoryIndex+13]
    Textfield (24,679 649x20), "%s", text variable: VAR_Explorer.Visu_Explorer.Directory[VAR_Explorer.Visu_Explorer.DirectoryIndex+14]
    Textfield (24,705 649x20), "%s", text variable: VAR_Explorer.Visu_Explorer.Directory[VAR_Explorer.Visu_Explorer.DirectoryIndex+15]
    Textfield (24,731 649x20), "%s", text variable: VAR_Explorer.Visu_Explorer.Directory[VAR_Explorer.Visu_Explorer.DirectoryIndex+16]
    Textfield (24,757 649x20), "%s", text variable: VAR_Explorer.Visu_Explorer.Directory[VAR_Explorer.Visu_Explorer.DirectoryIndex+17]
    Textfield (24,783 649x20), "%s", text variable: VAR_Explorer.Visu_Explorer.Directory[VAR_Explorer.Visu_Explorer.DirectoryIndex+18]
    Textfield (24,809 649x20), "%s", text variable: VAR_Explorer.Visu_Explorer.Directory[VAR_Explorer.Visu_Explorer.DirectoryIndex+19]
    Textfield (24,835 649x20), "%s", text variable: VAR_Explorer.Visu_Explorer.Directory[VAR_Explorer.Visu_Explorer.DirectoryIndex+20]
    Textfield (24,861 649x20), "%s", text variable: VAR_Explorer.Visu_Explorer.Directory[VAR_Explorer.Visu_Explorer.DirectoryIndex+21]
    Textfield (24,887 649x20), "%s", text variable: VAR_Explorer.Visu_Explorer.Directory[VAR_Explorer.Visu_Explorer.DirectoryIndex+22]
    Textfield (24,913 649x20), "%s", text variable: VAR_Explorer.Visu_Explorer.Directory[VAR_Explorer.Visu_Explorer.DirectoryIndex+23]
    Textfield (24,939 649x20), "%s", text variable: VAR_Explorer.Visu_Explorer.Directory[VAR_Explorer.Visu_Explorer.DirectoryIndex+24]
    Textfield (24,965 649x20), "%s", text variable: VAR_Explorer.Visu_Explorer.Directory[VAR_Explorer.Visu_Explorer.DirectoryIndex+25]
    Textfield (24,991 649x20), "%s", text variable: VAR_Explorer.Visu_Explorer.Directory[VAR_Explorer.Visu_Explorer.DirectoryIndex+26]
    Textfield (24,1017 649x20), "%s", text variable: VAR_Explorer.Visu_Explorer.Directory[VAR_Explorer.Visu_Explorer.DirectoryIndex+27]
    Textfield (24,1043 649x20), "%s", text variable: VAR_Explorer.Visu_Explorer.Directory[VAR_Explorer.Visu_Explorer.DirectoryIndex+28]
    Textfield (24,1069 649x20), "%s", text variable: VAR_Explorer.Visu_Explorer.Directory[VAR_Explorer.Visu_Explorer.DirectoryIndex+29]
    Textfield (24,1095 649x20), "%s", text variable: VAR_Explorer.Visu_Explorer.Directory[VAR_Explorer.Visu_Explorer.DirectoryIndex+30]
    Textfield (24,1121 649x20), "%s", text variable: VAR_Explorer.Visu_Explorer.Directory[VAR_Explorer.Visu_Explorer.DirectoryIndex+31]
    Button (949,315 100x20), "Ordner hoch"
        OnMouseUp: execute { VAR_Explorer.Visu_Explorer.folderUp := TRUE; }
    Group (691,315 100x826)
        Button (0,0 100x20), "Öffnen", invisible if: VAR_Explorer.Visu_Explorer.xdir[VAR_Explorer.Visu_Explorer.DirectoryIndex+0]
            OnMouseUp: execute { VAR_Explorer.Visu_Explorer.open := TRUE; VAR_Explorer.Visu_Explorer.openIndex := VAR_Explorer.Visu_Explorer.DirectoryIndex+0; }
        Button (0,26 100x20), "Öffnen", invisible if: VAR_Explorer.Visu_Explorer.xdir[VAR_Explorer.Visu_Explorer.DirectoryIndex+1]
            OnMouseUp: execute { VAR_Explorer.Visu_Explorer.open := TRUE; VAR_Explorer.Visu_Explorer.openIndex := VAR_Explorer.Visu_Explorer.DirectoryIndex+1; }
        Button (0,52 100x20), "Öffnen", invisible if: VAR_Explorer.Visu_Explorer.xdir[VAR_Explorer.Visu_Explorer.DirectoryIndex+2]
            OnMouseUp: execute { VAR_Explorer.Visu_Explorer.open := TRUE; VAR_Explorer.Visu_Explorer.openIndex := VAR_Explorer.Visu_Explorer.DirectoryIndex+2; }
        Button (0,78 100x20), "Öffnen", invisible if: VAR_Explorer.Visu_Explorer.xdir[VAR_Explorer.Visu_Explorer.DirectoryIndex+3]
            OnMouseUp: execute { VAR_Explorer.Visu_Explorer.open := TRUE; VAR_Explorer.Visu_Explorer.openIndex := VAR_Explorer.Visu_Explorer.DirectoryIndex+3; }
        Button (0,806 100x20), "Öffnen", invisible if: VAR_Explorer.Visu_Explorer.xdir[VAR_Explorer.Visu_Explorer.DirectoryIndex+31]
            OnMouseUp: execute { VAR_Explorer.Visu_Explorer.open := TRUE; VAR_Explorer.Visu_Explorer.openIndex := VAR_Explorer.Visu_Explorer.DirectoryIndex+31; }
        Button (0,104 100x20), "Öffnen", invisible if: VAR_Explorer.Visu_Explorer.xdir[VAR_Explorer.Visu_Explorer.DirectoryIndex+4]
            OnMouseUp: execute { VAR_Explorer.Visu_Explorer.open := TRUE; VAR_Explorer.Visu_Explorer.openIndex := VAR_Explorer.Visu_Explorer.DirectoryIndex+4; }
        Button (0,130 100x20), "Öffnen", invisible if: VAR_Explorer.Visu_Explorer.xdir[VAR_Explorer.Visu_Explorer.DirectoryIndex+5]
            OnMouseUp: execute { VAR_Explorer.Visu_Explorer.open := TRUE; VAR_Explorer.Visu_Explorer.openIndex := VAR_Explorer.Visu_Explorer.DirectoryIndex+5; }
        Button (0,156 100x20), "Öffnen", invisible if: VAR_Explorer.Visu_Explorer.xdir[VAR_Explorer.Visu_Explorer.DirectoryIndex+6]
            OnMouseUp: execute { VAR_Explorer.Visu_Explorer.open := TRUE; VAR_Explorer.Visu_Explorer.openIndex := VAR_Explorer.Visu_Explorer.DirectoryIndex+6; }
        Button (0,182 100x20), "Öffnen", invisible if: VAR_Explorer.Visu_Explorer.xdir[VAR_Explorer.Visu_Explorer.DirectoryIndex+7]
            OnMouseUp: execute { VAR_Explorer.Visu_Explorer.open := TRUE; VAR_Explorer.Visu_Explorer.openIndex := VAR_Explorer.Visu_Explorer.DirectoryIndex+7; }
        Button (0,208 100x20), "Öffnen", invisible if: VAR_Explorer.Visu_Explorer.xdir[VAR_Explorer.Visu_Explorer.DirectoryIndex+8]
            OnMouseUp: execute { VAR_Explorer.Visu_Explorer.open := TRUE; VAR_Explorer.Visu_Explorer.openIndex := VAR_Explorer.Visu_Explorer.DirectoryIndex+8; }
        Button (0,234 100x20), "Öffnen", invisible if: VAR_Explorer.Visu_Explorer.xdir[VAR_Explorer.Visu_Explorer.DirectoryIndex+9]
            OnMouseUp: execute { VAR_Explorer.Visu_Explorer.open := TRUE; VAR_Explorer.Visu_Explorer.openIndex := VAR_Explorer.Visu_Explorer.DirectoryIndex+9; }
        Button (0,260 100x20), "Öffnen", invisible if: VAR_Explorer.Visu_Explorer.xdir[VAR_Explorer.Visu_Explorer.DirectoryIndex+10]
            OnMouseUp: execute { VAR_Explorer.Visu_Explorer.open := TRUE; VAR_Explorer.Visu_Explorer.openIndex := VAR_Explorer.Visu_Explorer.DirectoryIndex+10; }
        Button (0,286 100x20), "Öffnen", invisible if: VAR_Explorer.Visu_Explorer.xdir[VAR_Explorer.Visu_Explorer.DirectoryIndex+11]
            OnMouseUp: execute { VAR_Explorer.Visu_Explorer.open := TRUE; VAR_Explorer.Visu_Explorer.openIndex := VAR_Explorer.Visu_Explorer.DirectoryIndex+11; }
        Button (0,312 100x20), "Öffnen", invisible if: VAR_Explorer.Visu_Explorer.xdir[VAR_Explorer.Visu_Explorer.DirectoryIndex+12]
            OnMouseUp: execute { VAR_Explorer.Visu_Explorer.open := TRUE; VAR_Explorer.Visu_Explorer.openIndex := VAR_Explorer.Visu_Explorer.DirectoryIndex+12; }
        Button (0,338 100x20), "Öffnen", invisible if: VAR_Explorer.Visu_Explorer.xdir[VAR_Explorer.Visu_Explorer.DirectoryIndex+13]
            OnMouseUp: execute { VAR_Explorer.Visu_Explorer.open := TRUE; VAR_Explorer.Visu_Explorer.openIndex := VAR_Explorer.Visu_Explorer.DirectoryIndex+13; }
        Button (0,364 100x20), "Öffnen", invisible if: VAR_Explorer.Visu_Explorer.xdir[VAR_Explorer.Visu_Explorer.DirectoryIndex+14]
            OnMouseUp: execute { VAR_Explorer.Visu_Explorer.open := TRUE; VAR_Explorer.Visu_Explorer.openIndex := VAR_Explorer.Visu_Explorer.DirectoryIndex+14; }
        Button (0,390 100x20), "Öffnen", invisible if: VAR_Explorer.Visu_Explorer.xdir[VAR_Explorer.Visu_Explorer.DirectoryIndex+15]
            OnMouseUp: execute { VAR_Explorer.Visu_Explorer.open := TRUE; VAR_Explorer.Visu_Explorer.openIndex := VAR_Explorer.Visu_Explorer.DirectoryIndex+15; }
        Button (0,416 100x20), "Öffnen", invisible if: VAR_Explorer.Visu_Explorer.xdir[VAR_Explorer.Visu_Explorer.DirectoryIndex+16]
            OnMouseUp: execute { VAR_Explorer.Visu_Explorer.open := TRUE; VAR_Explorer.Visu_Explorer.openIndex := VAR_Explorer.Visu_Explorer.DirectoryIndex+16; }
        Button (0,442 100x20), "Öffnen", invisible if: VAR_Explorer.Visu_Explorer.xdir[VAR_Explorer.Visu_Explorer.DirectoryIndex+17]
            OnMouseUp: execute { VAR_Explorer.Visu_Explorer.open := TRUE; VAR_Explorer.Visu_Explorer.openIndex := VAR_Explorer.Visu_Explorer.DirectoryIndex+17; }
        Button (0,468 100x20), "Öffnen", invisible if: VAR_Explorer.Visu_Explorer.xdir[VAR_Explorer.Visu_Explorer.DirectoryIndex+18]
            OnMouseUp: execute { VAR_Explorer.Visu_Explorer.open := TRUE; VAR_Explorer.Visu_Explorer.openIndex := VAR_Explorer.Visu_Explorer.DirectoryIndex+18; }
        Button (0,494 100x20), "Öffnen", invisible if: VAR_Explorer.Visu_Explorer.xdir[VAR_Explorer.Visu_Explorer.DirectoryIndex+19]
            OnMouseUp: execute { VAR_Explorer.Visu_Explorer.open := TRUE; VAR_Explorer.Visu_Explorer.openIndex := VAR_Explorer.Visu_Explorer.DirectoryIndex+19; }
        Button (0,520 100x20), "Öffnen", invisible if: VAR_Explorer.Visu_Explorer.xdir[VAR_Explorer.Visu_Explorer.DirectoryIndex+20]
            OnMouseUp: execute { VAR_Explorer.Visu_Explorer.open := TRUE; VAR_Explorer.Visu_Explorer.openIndex := VAR_Explorer.Visu_Explorer.DirectoryIndex+20; }
        Button (0,546 100x20), "Öffnen", invisible if: VAR_Explorer.Visu_Explorer.xdir[VAR_Explorer.Visu_Explorer.DirectoryIndex+21]
            OnMouseUp: execute { VAR_Explorer.Visu_Explorer.open := TRUE; VAR_Explorer.Visu_Explorer.openIndex := VAR_Explorer.Visu_Explorer.DirectoryIndex+21; }
        Button (0,572 100x20), "Öffnen", invisible if: VAR_Explorer.Visu_Explorer.xdir[VAR_Explorer.Visu_Explorer.DirectoryIndex+22]
            OnMouseUp: execute { VAR_Explorer.Visu_Explorer.open := TRUE; VAR_Explorer.Visu_Explorer.openIndex := VAR_Explorer.Visu_Explorer.DirectoryIndex+22; }
        Button (0,598 100x20), "Öffnen", invisible if: VAR_Explorer.Visu_Explorer.xdir[VAR_Explorer.Visu_Explorer.DirectoryIndex+23]
            OnMouseUp: execute { VAR_Explorer.Visu_Explorer.open := TRUE; VAR_Explorer.Visu_Explorer.openIndex := VAR_Explorer.Visu_Explorer.DirectoryIndex+23; }
        Button (0,624 100x20), "Öffnen", invisible if: VAR_Explorer.Visu_Explorer.xdir[VAR_Explorer.Visu_Explorer.DirectoryIndex+24]
            OnMouseUp: execute { VAR_Explorer.Visu_Explorer.open := TRUE; VAR_Explorer.Visu_Explorer.openIndex := VAR_Explorer.Visu_Explorer.DirectoryIndex+24; }
        Button (0,650 100x20), "Öffnen", invisible if: VAR_Explorer.Visu_Explorer.xdir[VAR_Explorer.Visu_Explorer.DirectoryIndex+25]
            OnMouseUp: execute { VAR_Explorer.Visu_Explorer.open := TRUE; VAR_Explorer.Visu_Explorer.openIndex := VAR_Explorer.Visu_Explorer.DirectoryIndex+25; }
        Button (0,676 100x20), "Öffnen", invisible if: VAR_Explorer.Visu_Explorer.xdir[VAR_Explorer.Visu_Explorer.DirectoryIndex+26]
            OnMouseUp: execute { VAR_Explorer.Visu_Explorer.open := TRUE; VAR_Explorer.Visu_Explorer.openIndex := VAR_Explorer.Visu_Explorer.DirectoryIndex+26; }
        Button (0,702 100x20), "Öffnen", invisible if: VAR_Explorer.Visu_Explorer.xdir[VAR_Explorer.Visu_Explorer.DirectoryIndex+27]
            OnMouseUp: execute { VAR_Explorer.Visu_Explorer.open := TRUE; VAR_Explorer.Visu_Explorer.openIndex := VAR_Explorer.Visu_Explorer.DirectoryIndex+27; }
        Button (0,728 100x20), "Öffnen", invisible if: VAR_Explorer.Visu_Explorer.xdir[VAR_Explorer.Visu_Explorer.DirectoryIndex+28]
            OnMouseUp: execute { VAR_Explorer.Visu_Explorer.open := TRUE; VAR_Explorer.Visu_Explorer.openIndex := VAR_Explorer.Visu_Explorer.DirectoryIndex+28; }
        Button (0,754 100x20), "Öffnen", invisible if: VAR_Explorer.Visu_Explorer.xdir[VAR_Explorer.Visu_Explorer.DirectoryIndex+29]
            OnMouseUp: execute { VAR_Explorer.Visu_Explorer.open := TRUE; VAR_Explorer.Visu_Explorer.openIndex := VAR_Explorer.Visu_Explorer.DirectoryIndex+29; }
        Button (0,780 100x20), "Öffnen", invisible if: VAR_Explorer.Visu_Explorer.xdir[VAR_Explorer.Visu_Explorer.DirectoryIndex+30]
            OnMouseUp: execute { VAR_Explorer.Visu_Explorer.open := TRUE; VAR_Explorer.Visu_Explorer.openIndex := VAR_Explorer.Visu_Explorer.DirectoryIndex+30; }
    Textfield (24,281 1090x20), "%s", text variable: VAR_Explorer.Visu_Explorer.actualsharePath
    Rectangle (439,66 150x25), "Conntected", invisible if: VAR_Explorer.Visu_Explorer.online
    Rectangle (606,66 150x25), "Error", invisible if: VAR_Explorer.Visu_Explorer.error
    Button (819,315 38x20), "hoch"
        OnMouseUp: execute {
            VAR_Explorer.Visu_Explorer.DirectoryIndex:=VAR_Explorer.Visu_Explorer.DirectoryIndex-5;
            IF VAR_Explorer.Visu_Explorer.DirectoryIndex <=0 THEN
            	VAR_Explorer.Visu_Explorer.DirectoryIndex:=0;
            END_IF
        }
    Button (819,1121 38x20), "runter"
        OnMouseUp: execute {
            VAR_Explorer.Visu_Explorer.DirectoryIndex:=VAR_Explorer.Visu_Explorer.DirectoryIndex+5;
            IF VAR_Explorer.Visu_Explorer.DirectoryIndex >=128 THEN
            	VAR_Explorer.Visu_Explorer.DirectoryIndex:=128;
            END_IF
        }
    Textfield (25,163 1090x20), "%s", text variable: VAR_Explorer.Visu_Explorer.copysharePath
        OnMouseDown: write the text variable via Edit
    Label (27,136 264x30), "Pfad für automatische Übertragung"
    Label (29,250 116x30), "Aktueller Pfad"
    Group (691,315 100x826)
        Button (0,0 100x20), "Übernehmen", invisible if: VAR_Explorer.Visu_Explorer.xfile[VAR_Explorer.Visu_Explorer.DirectoryIndex+0]
            OnMouseUp: execute { VAR_Explorer.Visu_Explorer.apply := TRUE; VAR_Explorer.Visu_Explorer.applyIndex := VAR_Explorer.Visu_Explorer.DirectoryIndex+0; }
        Button (0,26 100x20), "Übernehmen", invisible if: VAR_Explorer.Visu_Explorer.xfile[VAR_Explorer.Visu_Explorer.DirectoryIndex+1]
            OnMouseUp: execute { VAR_Explorer.Visu_Explorer.apply := TRUE; VAR_Explorer.Visu_Explorer.applyIndex := VAR_Explorer.Visu_Explorer.DirectoryIndex+1; }
        Button (0,52 100x20), "Übernehmen", invisible if: VAR_Explorer.Visu_Explorer.xfile[VAR_Explorer.Visu_Explorer.DirectoryIndex+2]
            OnMouseUp: execute { VAR_Explorer.Visu_Explorer.apply := TRUE; VAR_Explorer.Visu_Explorer.applyIndex := VAR_Explorer.Visu_Explorer.DirectoryIndex+2; }
        Button (0,78 100x20), "Übernehmen", invisible if: VAR_Explorer.Visu_Explorer.xfile[VAR_Explorer.Visu_Explorer.DirectoryIndex+3]
            OnMouseUp: execute { VAR_Explorer.Visu_Explorer.apply := TRUE; VAR_Explorer.Visu_Explorer.applyIndex := VAR_Explorer.Visu_Explorer.DirectoryIndex+3; }
        Button (0,806 100x20), "Übernehmen", invisible if: VAR_Explorer.Visu_Explorer.xfile[VAR_Explorer.Visu_Explorer.DirectoryIndex+31]
            OnMouseUp: execute { VAR_Explorer.Visu_Explorer.apply := TRUE; VAR_Explorer.Visu_Explorer.applyIndex := VAR_Explorer.Visu_Explorer.DirectoryIndex+31; }
        Button (0,104 100x20), "Übernehmen", invisible if: VAR_Explorer.Visu_Explorer.xfile[VAR_Explorer.Visu_Explorer.DirectoryIndex+4]
            OnMouseUp: execute { VAR_Explorer.Visu_Explorer.apply := TRUE; VAR_Explorer.Visu_Explorer.applyIndex := VAR_Explorer.Visu_Explorer.DirectoryIndex+4; }
        Button (0,130 100x20), "Übernehmen", invisible if: VAR_Explorer.Visu_Explorer.xfile[VAR_Explorer.Visu_Explorer.DirectoryIndex+5]
            OnMouseUp: execute { VAR_Explorer.Visu_Explorer.apply := TRUE; VAR_Explorer.Visu_Explorer.applyIndex := VAR_Explorer.Visu_Explorer.DirectoryIndex+5; }
        Button (0,156 100x20), "Übernehmen", invisible if: VAR_Explorer.Visu_Explorer.xfile[VAR_Explorer.Visu_Explorer.DirectoryIndex+6]
            OnMouseUp: execute { VAR_Explorer.Visu_Explorer.apply := TRUE; VAR_Explorer.Visu_Explorer.applyIndex := VAR_Explorer.Visu_Explorer.DirectoryIndex+6; }
        Button (0,182 100x20), "Übernehmen", invisible if: VAR_Explorer.Visu_Explorer.xfile[VAR_Explorer.Visu_Explorer.DirectoryIndex+7]
            OnMouseUp: execute { VAR_Explorer.Visu_Explorer.apply := TRUE; VAR_Explorer.Visu_Explorer.applyIndex := VAR_Explorer.Visu_Explorer.DirectoryIndex+7; }
        Button (0,208 100x20), "Übernehmen", invisible if: VAR_Explorer.Visu_Explorer.xfile[VAR_Explorer.Visu_Explorer.DirectoryIndex+8]
            OnMouseUp: execute { VAR_Explorer.Visu_Explorer.apply := TRUE; VAR_Explorer.Visu_Explorer.applyIndex := VAR_Explorer.Visu_Explorer.DirectoryIndex+8; }
        Button (0,234 100x20), "Übernehmen", invisible if: VAR_Explorer.Visu_Explorer.xfile[VAR_Explorer.Visu_Explorer.DirectoryIndex+9]
            OnMouseUp: execute { VAR_Explorer.Visu_Explorer.apply := TRUE; VAR_Explorer.Visu_Explorer.applyIndex := VAR_Explorer.Visu_Explorer.DirectoryIndex+9; }
        Button (0,260 100x20), "Übernehmen", invisible if: VAR_Explorer.Visu_Explorer.xfile[VAR_Explorer.Visu_Explorer.DirectoryIndex+10]
            OnMouseUp: execute { VAR_Explorer.Visu_Explorer.apply := TRUE; VAR_Explorer.Visu_Explorer.applyIndex := VAR_Explorer.Visu_Explorer.DirectoryIndex+10; }
        Button (0,286 100x20), "Übernehmen", invisible if: VAR_Explorer.Visu_Explorer.xfile[VAR_Explorer.Visu_Explorer.DirectoryIndex+11]
            OnMouseUp: execute { VAR_Explorer.Visu_Explorer.apply := TRUE; VAR_Explorer.Visu_Explorer.applyIndex := VAR_Explorer.Visu_Explorer.DirectoryIndex+11; }
        Button (0,312 100x20), "Übernehmen", invisible if: VAR_Explorer.Visu_Explorer.xfile[VAR_Explorer.Visu_Explorer.DirectoryIndex+12]
            OnMouseUp: execute { VAR_Explorer.Visu_Explorer.apply := TRUE; VAR_Explorer.Visu_Explorer.applyIndex := VAR_Explorer.Visu_Explorer.DirectoryIndex+12; }
        Button (0,338 100x20), "Übernehmen", invisible if: VAR_Explorer.Visu_Explorer.xfile[VAR_Explorer.Visu_Explorer.DirectoryIndex+13]
            OnMouseUp: execute { VAR_Explorer.Visu_Explorer.apply := TRUE; VAR_Explorer.Visu_Explorer.applyIndex := VAR_Explorer.Visu_Explorer.DirectoryIndex+13; }
        Button (0,364 100x20), "Übernehmen", invisible if: VAR_Explorer.Visu_Explorer.xfile[VAR_Explorer.Visu_Explorer.DirectoryIndex+14]
            OnMouseUp: execute { VAR_Explorer.Visu_Explorer.apply := TRUE; VAR_Explorer.Visu_Explorer.applyIndex := VAR_Explorer.Visu_Explorer.DirectoryIndex+14; }
        Button (0,390 100x20), "Übernehmen", invisible if: VAR_Explorer.Visu_Explorer.xfile[VAR_Explorer.Visu_Explorer.DirectoryIndex+15]
            OnMouseUp: execute { VAR_Explorer.Visu_Explorer.apply := TRUE; VAR_Explorer.Visu_Explorer.applyIndex := VAR_Explorer.Visu_Explorer.DirectoryIndex+15; }
        Button (0,416 100x20), "Übernehmen", invisible if: VAR_Explorer.Visu_Explorer.xfile[VAR_Explorer.Visu_Explorer.DirectoryIndex+16]
            OnMouseUp: execute { VAR_Explorer.Visu_Explorer.apply := TRUE; VAR_Explorer.Visu_Explorer.applyIndex := VAR_Explorer.Visu_Explorer.DirectoryIndex+16; }
        Button (0,442 100x20), "Übernehmen", invisible if: VAR_Explorer.Visu_Explorer.xfile[VAR_Explorer.Visu_Explorer.DirectoryIndex+17]
            OnMouseUp: execute { VAR_Explorer.Visu_Explorer.apply := TRUE; VAR_Explorer.Visu_Explorer.applyIndex := VAR_Explorer.Visu_Explorer.DirectoryIndex+17; }
        Button (0,468 100x20), "Übernehmen", invisible if: VAR_Explorer.Visu_Explorer.xfile[VAR_Explorer.Visu_Explorer.DirectoryIndex+18]
            OnMouseUp: execute { VAR_Explorer.Visu_Explorer.apply := TRUE; VAR_Explorer.Visu_Explorer.applyIndex := VAR_Explorer.Visu_Explorer.DirectoryIndex+18; }
        Button (0,494 100x20), "Übernehmen", invisible if: VAR_Explorer.Visu_Explorer.xfile[VAR_Explorer.Visu_Explorer.DirectoryIndex+19]
            OnMouseUp: execute { VAR_Explorer.Visu_Explorer.apply := TRUE; VAR_Explorer.Visu_Explorer.applyIndex := VAR_Explorer.Visu_Explorer.DirectoryIndex+19; }
        Button (0,520 100x20), "Übernehmen", invisible if: VAR_Explorer.Visu_Explorer.xfile[VAR_Explorer.Visu_Explorer.DirectoryIndex+20]
            OnMouseUp: execute { VAR_Explorer.Visu_Explorer.apply := TRUE; VAR_Explorer.Visu_Explorer.applyIndex := VAR_Explorer.Visu_Explorer.DirectoryIndex+20; }
        Button (0,546 100x20), "Übernehmen", invisible if: VAR_Explorer.Visu_Explorer.xfile[VAR_Explorer.Visu_Explorer.DirectoryIndex+21]
            OnMouseUp: execute { VAR_Explorer.Visu_Explorer.apply := TRUE; VAR_Explorer.Visu_Explorer.applyIndex := VAR_Explorer.Visu_Explorer.DirectoryIndex+21; }
        Button (0,572 100x20), "Übernehmen", invisible if: VAR_Explorer.Visu_Explorer.xfile[VAR_Explorer.Visu_Explorer.DirectoryIndex+22]
            OnMouseUp: execute { VAR_Explorer.Visu_Explorer.apply := TRUE; VAR_Explorer.Visu_Explorer.applyIndex := VAR_Explorer.Visu_Explorer.DirectoryIndex+22; }
        Button (0,598 100x20), "Übernehmen", invisible if: VAR_Explorer.Visu_Explorer.xfile[VAR_Explorer.Visu_Explorer.DirectoryIndex+23]
            OnMouseUp: execute { VAR_Explorer.Visu_Explorer.apply := TRUE; VAR_Explorer.Visu_Explorer.applyIndex := VAR_Explorer.Visu_Explorer.DirectoryIndex+23; }
        Button (0,624 100x20), "Übernehmen", invisible if: VAR_Explorer.Visu_Explorer.xfile[VAR_Explorer.Visu_Explorer.DirectoryIndex+24]
            OnMouseUp: execute { VAR_Explorer.Visu_Explorer.apply := TRUE; VAR_Explorer.Visu_Explorer.applyIndex := VAR_Explorer.Visu_Explorer.DirectoryIndex+24; }
        Button (0,650 100x20), "Übernehmen", invisible if: VAR_Explorer.Visu_Explorer.xfile[VAR_Explorer.Visu_Explorer.DirectoryIndex+25]
            OnMouseUp: execute { VAR_Explorer.Visu_Explorer.apply := TRUE; VAR_Explorer.Visu_Explorer.applyIndex := VAR_Explorer.Visu_Explorer.DirectoryIndex+25; }
        Button (0,676 100x20), "Übernehmen", invisible if: VAR_Explorer.Visu_Explorer.xfile[VAR_Explorer.Visu_Explorer.DirectoryIndex+26]
            OnMouseUp: execute { VAR_Explorer.Visu_Explorer.apply := TRUE; VAR_Explorer.Visu_Explorer.applyIndex := VAR_Explorer.Visu_Explorer.DirectoryIndex+26; }
        Button (0,702 100x20), "Übernehmen", invisible if: VAR_Explorer.Visu_Explorer.xfile[VAR_Explorer.Visu_Explorer.DirectoryIndex+27]
            OnMouseUp: execute { VAR_Explorer.Visu_Explorer.apply := TRUE; VAR_Explorer.Visu_Explorer.applyIndex := VAR_Explorer.Visu_Explorer.DirectoryIndex+27; }
        Button (0,728 100x20), "Übernehmen", invisible if: VAR_Explorer.Visu_Explorer.xfile[VAR_Explorer.Visu_Explorer.DirectoryIndex+28]
            OnMouseUp: execute { VAR_Explorer.Visu_Explorer.apply := TRUE; VAR_Explorer.Visu_Explorer.applyIndex := VAR_Explorer.Visu_Explorer.DirectoryIndex+28; }
        Button (0,754 100x20), "Übernehmen", invisible if: VAR_Explorer.Visu_Explorer.xfile[VAR_Explorer.Visu_Explorer.DirectoryIndex+29]
            OnMouseUp: execute { VAR_Explorer.Visu_Explorer.apply := TRUE; VAR_Explorer.Visu_Explorer.applyIndex := VAR_Explorer.Visu_Explorer.DirectoryIndex+29; }
        Button (0,780 100x20), "Übernehmen", invisible if: VAR_Explorer.Visu_Explorer.xfile[VAR_Explorer.Visu_Explorer.DirectoryIndex+30]
            OnMouseUp: execute { VAR_Explorer.Visu_Explorer.apply := TRUE; VAR_Explorer.Visu_Explorer.applyIndex := VAR_Explorer.Visu_Explorer.DirectoryIndex+30; }
    Textfield (25,213 1090x20), "%s", text variable: VAR_Explorer.Visu_Explorer.plcPath
        OnMouseDown: write the text variable via Edit
    Label (27,186 111x30), "Pfad auf PLC"
    Rectangle (765,66 68x25), "Busy", invisible if: VAR_Explorer.Visu_Explorer.busy
    Rectangle (842,66 68x25), "Done", invisible if: VAR_Explorer.Visu_Explorer.done
    Button (930,32 100x25), "SPS -> PC", colour toggle: VAR_Explorer.Visu_Explorer.write
        OnMouseUp: execute {
            VAR_Explorer.Visu_Explorer.write_read := 1;
            VAR_Explorer.Visu_Explorer.write := TRUE;
            VAR_Explorer.Visu_Explorer.read := FALSE;
        }
    Button (930,66 100x25), "PC -> SPS", colour toggle: VAR_Explorer.Visu_Explorer.read
        OnMouseUp: execute {
            VAR_Explorer.Visu_Explorer.write_read := 2;
            VAR_Explorer.Visu_Explorer.write := FALSE;
            VAR_Explorer.Visu_Explorer.read := TRUE;
        }
    Button (1043,32 100x60), "Start Übertragung"
        tap VAR_Explorer.Visu_Explorer.start
    Label (1145,39 131x76), "Zum starten der Übertragung erst ausloggen"
END_VISUALIZATION
